C09025=1038.692,60.769,-88.501,169.467,39.132,157.356
C09026=1038.685,60.483,-88.481,169.465,39.132,157.356
C09027=1038.677,60.197,-88.461,169.463,39.132,157.356
C09028=1038.672,59.947,-88.444,169.461,39.131,157.356
C09029=1038.665,59.698,-88.426,169.459,39.131,157.356
C09030=1038.659,59.448,-88.409,169.457,39.131,157.356
C09031=1038.652,59.200,-88.392,169.454,39.130,157.356
C09032=1038.645,58.951,-88.373,169.452,39.130,157.356
C09033=1038.639,58.701,-88.356,169.450,39.130,157.355
C09034=1038.633,58.452,-88.339,169.448,39.129,157.355
C09035=1038.627,58.203,-88.321,169.446,39.130,157.355
C09036=1038.620,57.953,-88.303,169.444,39.129,157.355
C09037=1038.614,57.704,-88.286,169.442,39.129,157.355
C09038=1038.607,57.455,-88.268,169.440,39.128,157.355
C09039=1038.601,57.205,-88.251,169.438,39.128,157.355
C09040=1038.594,56.956,-88.234,169.436,39.128,157.355
C09041=1038.589,56.706,-88.217,169.433,39.127,157.354
C09042=1038.582,56.457,-88.200,169.432,39.127,157.354
C09043=1038.575,56.208,-88.183,169.430,39.127,157.354
C09044=1038.569,55.958,-88.165,169.428,39.126,157.354
C09045=1038.562,55.709,-88.147,169.426,39.126,157.354
C09046=1038.557,55.460,-88.130,169.424,39.126,157.354
C09047=1038.550,55.210,-88.112,169.422,39.125,157.354
C09048=1038.544,54.962,-88.095,169.420,39.125,157.354
C09049=1038.538,54.712,-88.077,169.418,39.125,157.354
C09050=1038.531,54.462,-88.060,169.416,39.125,157.353
C09051=1038.525,54.214,-88.043,169.413,39.124,157.353
C09052=1038.518,53.964,-88.025,169.411,39.124,157.353
C09053=1038.512,53.715,-88.008,169.409,39.124,157.353
C09054=1038.506,53.465,-87.992,169.407,39.123,157.353
C09055=1038.500,53.216,-87.974,169.405,39.123,157.353
C09056=1038.493,52.967,-87.957,169.404,39.123,157.353
C09057=1038.486,52.717,-87.939,169.402,39.122,157.353
C09058=1038.481,52.468,-87.922,169.400,39.122,157.352
C09059=1038.474,52.219,-87.905,169.398,39.121,157.352
C09060=1038.468,51.970,-87.888,169.395,39.121,157.352
C09061=1038.462,51.720,-87.870,169.393,39.121,157.352
C09062=1038.456,51.471,-87.853,169.391,39.120,157.352
C09063=1038.449,51.222,-87.836,169.389,39.120,157.352
C09064=1038.443,50.973,-87.818,169.387,39.120,157.352
C09065=1038.437,50.723,-87.801,169.385,39.119,157.352
C09066=1038.431,50.474,-87.785,169.383,39.119,157.351
C09067=1038.424,50.224,-87.767,169.381,39.119,157.351
C09068=1038.418,49.975,-87.750,169.379,39.119,157.351
C09069=1038.411,49.726,-87.733,169.378,39.118,157.351
C09070=1038.406,49.475,-87.715,169.375,39.118,157.351
C09071=1038.399,49.227,-87.698,169.373,39.118,157.351
C09072=1038.393,48.978,-87.681,169.371,39.117,157.351
C09073=1038.387,48.728,-87.664,169.369,39.117,157.351
C09074=1038.381,48.479,-87.647,169.367,39.116,157.350
C09075=1038.374,48.230,-87.630,169.365,39.116,157.350
C09076=1038.369,47.980,-87.612,169.363,39.116,157.350
C09077=1038.362,47.731,-87.595,169.361,39.115,157.350
C09078=1038.356,47.482,-87.579,169.359,39.115,157.350
C09079=1038.350,47.232,-87.561,169.356,39.114,157.350
C09080=1038.343,46.983,-87.544,169.354,39.114,157.350
C09081=1038.337,46.733,-87.527,169.352,39.114,157.350
C09082=1038.331,46.484,-87.510,169.351,39.113,157.349
C09083=1038.324,46.235,-87.492,169.349,39.113,157.349
C09084=1038.318,45.985,-87.476,169.347,39.112,157.349
C09085=1038.312,45.737,-87.459,169.345,39.112,157.349
C09086=1038.306,45.487,-87.441,169.343,39.112,157.349
C09087=1038.300,45.238,-87.425,169.341,39.111,157.349
C09088=1038.293,44.951,-87.405,169.338,39.111,157.349
C09089=1038.286,44.664,-87.385,169.336,39.110,157.348
C09090=1038.279,44.378,-87.366,169.333,39.110,157.348
C09091=1038.271,44.091,-87.346,169.331,39.109,157.348
C09092=1038.266,43.842,-87.330,169.329,39.110,157.348
C09093=1038.259,43.592,-87.312,169.327,39.109,157.348
C09094=1038.253,43.343,-87.296,169.325,39.109,157.348
C09095=1038.247,43.094,-87.278,169.323,39.108,157.348
C09096=1038.241,42.845,-87.261,169.321,39.108,157.348
C09097=1038.235,42.595,-87.245,169.319,39.108,157.347
C09098=1038.228,42.346,-87.227,169.317,39.107,157.347
C09099=1038.222,42.096,-87.211,169.315,39.107,157.347
C09100=1038.215,41.846,-87.195,169.313,39.107,157.347
C09101=1038.209,41.598,-87.178,169.311,39.106,157.347
C09102=1038.203,41.348,-87.161,169.309,39.106,157.347
C09103=1038.196,41.099,-87.144,169.307,39.106,157.347
C09104=1038.190,40.849,-87.128,169.305,39.105,157.347
C09105=1038.183,40.600,-87.110,169.303,39.105,157.347
C09106=1038.177,40.351,-87.094,169.301,39.105,157.346
C09107=1038.171,40.102,-87.077,169.298,39.104,157.346
C09108=1038.165,39.852,-87.061,169.296,39.105,157.346
C09109=1038.159,39.603,-87.044,169.294,39.104,157.346
C09110=1038.152,39.354,-87.027,169.292,39.104,157.346
C09111=1038.146,39.104,-87.011,169.290,39.104,157.346
C09112=1038.140,38.855,-86.994,169.288,39.103,157.346
C09113=1038.133,38.605,-86.977,169.286,39.103,157.346
C09114=1038.127,38.356,-86.961,169.284,39.103,157.346
C09115=1038.121,38.107,-86.944,169.282,39.102,157.345
C09116=1038.114,37.857,-86.927,169.279,39.102,157.345
C09117=1038.108,37.608,-86.911,169.277,39.102,157.345
C09118=1038.102,37.359,-86.894,169.275,39.101,157.345
C09119=1038.096,37.109,-86.877,169.273,39.101,157.345
C09120=1038.090,36.859,-86.861,169.271,39.101,157.345
C09121=1038.083,36.611,-86.844,169.269,39.101,157.345
C09122=1038.076,36.361,-86.828,169.267,39.101,157.345
C09123=1038.070,36.112,-86.812,169.265,39.100,157.344
C09124=1038.064,35.862,-86.796,169.263,39.100,157.344
C09125=1038.057,35.613,-86.778,169.261,39.100,157.344
C09126=1038.051,35.363,-86.762,169.259,39.099,157.344
C09127=1038.045,35.114,-86.746,169.257,39.099,157.344
C09128=1038.038,34.864,-86.730,169.255,39.099,157.344
C09129=1038.032,34.616,-86.713,169.253,39.099,157.344
C09130=1038.026,34.366,-86.697,169.251,39.099,157.344
C09131=1038.019,34.116,-86.680,169.249,39.098,157.344
C09132=1038.013,33.867,-86.664,169.247,39.098,157.344
C09133=1038.007,33.618,-86.648,169.245,39.098,157.343
C09134=1038.000,33.368,-86.631,169.243,39.098,157.343
C09135=1037.994,33.119,-86.614,169.241,39.097,157.343
C09136=1037.988,32.870,-86.598,169.239,39.097,157.343
C09137=1037.981,32.620,-86.582,169.237,39.097,157.343
C09138=1037.975,32.371,-86.566,169.235,39.096,157.343
C09139=1037.969,32.121,-86.550,169.233,39.097,157.343
C09140=1037.962,31.873,-86.533,169.230,39.096,157.343
C09141=1037.956,31.623,-86.516,169.228,39.095,157.343
C09142=1037.949,31.374,-86.500,169.226,39.096,157.342
C09143=1037.943,31.124,-86.484,169.224,39.095,157.342
C09144=1037.937,30.875,-86.468,169.222,39.095,157.342
C09145=1037.931,30.625,-86.451,169.220,39.095,157.342
C09146=1037.924,30.376,-86.436,169.218,39.094,157.342
C09147=1037.918,30.126,-86.419,169.216,39.094,157.342
C09148=1037.912,29.877,-86.403,169.214,39.094,157.342
C09149=1037.906,29.627,-86.386,169.212,39.094,157.342
C09150=1037.899,29.379,-86.370,169.210,39.093,157.342
C09151=1037.893,29.129,-86.354,169.207,39.093,157.341
C09152=1037.886,28.842,-86.336,169.204,39.093,157.341
C09153=1037.879,28.556,-86.317,169.202,39.093,157.341
C09154=1037.871,28.269,-86.298,169.200,39.092,157.341
C09155=1037.864,27.982,-86.280,169.197,39.092,157.341
C09156=1037.858,27.733,-86.263,169.195,39.092,157.341
C09157=1037.851,27.484,-86.248,169.193,39.092,157.341
C09158=1037.845,27.234,-86.231,169.191,39.091,157.341
C09159=1037.839,26.984,-86.215,169.189,39.091,157.341
C09160=1037.832,26.735,-86.199,169.187,39.091,157.340
C09161=1037.826,26.486,-86.183,169.184,39.091,157.340
C09162=1037.819,26.237,-86.167,169.182,39.091,157.340
C09163=1037.813,25.987,-86.151,169.180,39.090,157.340
C09164=1037.806,25.738,-86.135,169.178,39.090,157.340
C09165=1037.800,25.488,-86.119,169.176,39.090,157.340
C09166=1037.794,25.239,-86.102,169.174,39.090,157.340
C09167=1037.788,24.989,-86.088,169.172,39.089,157.340
C09168=1037.781,24.739,-86.071,169.170,39.090,157.340
C09169=1037.775,24.490,-86.055,169.168,39.089,157.340
C09170=1037.769,24.241,-86.039,169.166,39.089,157.340
C09171=1037.762,23.992,-86.023,169.164,39.089,157.339
C09172=1037.756,23.742,-86.007,169.162,39.089,157.339
C09173=1037.749,23.493,-85.991,169.160,39.088,157.339
C09174=1037.743,23.243,-85.976,169.158,39.088,157.339
C09175=1037.736,22.994,-85.960,169.155,39.088,157.339
C09176=1037.730,22.744,-85.944,169.153,39.088,157.339
C09177=1037.724,22.495,-85.928,169.151,39.088,157.339
C09178=1037.718,22.246,-85.912,169.149,39.088,157.339
C09179=1037.711,21.997,-85.896,169.147,39.087,157.339
C09180=1037.705,21.747,-85.880,169.145,39.087,157.338
C09181=1037.699,21.498,-85.865,169.143,39.087,157.338
C09182=1037.692,21.248,-85.848,169.141,39.086,157.338
C09183=1037.686,20.999,-85.833,169.139,39.086,157.338
C09184=1037.680,20.749,-85.817,169.137,39.086,157.338
C09185=1037.673,20.500,-85.801,169.135,39.086,157.338
C09186=1037.667,20.251,-85.785,169.133,39.086,157.338
C09187=1037.661,20.001,-85.769,169.129,39.086,157.338
C09188=1037.655,19.752,-85.754,169.127,39.085,157.338
C09189=1037.648,19.502,-85.738,169.125,39.085,157.338
C09190=1037.642,19.253,-85.722,169.123,39.085,157.338
C09191=1037.635,19.003,-85.707,169.121,39.085,157.337
C09192=1037.629,18.753,-85.690,169.119,39.084,157.337
C09193=1037.623,18.504,-85.675,169.117,39.085,157.337
C09194=1037.616,18.255,-85.660,169.115,39.084,157.337
C09195=1037.610,18.005,-85.644,169.113,39.084,157.337
C09196=1037.604,17.756,-85.628,169.111,39.084,157.337
C09197=1037.597,17.507,-85.613,169.109,39.084,157.337
C09198=1037.591,17.257,-85.597,169.107,39.083,157.337
C09199=1037.585,17.008,-85.581,169.105,39.083,157.337
C09200=1037.578,16.759,-85.566,169.102,39.083,157.337
C09201=1037.572,16.509,-85.550,169.100,39.083,157.337
C09202=1037.566,16.260,-85.535,169.098,39.083,157.336
C09203=1037.560,16.010,-85.519,169.096,39.083,157.336
C09204=1037.553,15.761,-85.503,169.093,39.082,157.336
C09205=1037.547,15.512,-85.488,169.091,39.082,157.336
C09206=1037.541,15.262,-85.472,169.089,39.082,157.336
C09207=1037.535,15.013,-85.457,169.087,39.082,157.336
C09208=1037.527,14.763,-85.441,169.085,39.082,157.336
C09209=1037.522,14.513,-85.425,169.083,39.082,157.336
C09210=1037.515,14.264,-85.410,169.081,39.082,157.336
C09211=1037.509,14.014,-85.395,169.079,39.081,157.336
C09212=1037.503,13.765,-85.378,169.077,39.081,157.336
C09213=1037.496,13.515,-85.363,169.074,39.081,157.335
C09214=1037.490,13.266,-85.348,169.072,39.081,157.335
C09215=1037.483,13.016,-85.333,169.070,39.081,157.335
C09216=1037.476,12.731,-85.315,169.067,39.081,157.335
C09217=1037.468,12.446,-85.297,169.065,39.081,157.335
C09218=1037.461,12.161,-85.280,169.062,39.080,157.335
C09219=1037.454,11.876,-85.263,169.060,39.081,157.335
C09220=1037.447,11.626,-85.247,169.058,39.081,157.335
C09221=1037.440,11.376,-85.232,169.056,39.080,157.335
C09222=1037.434,11.127,-85.217,169.054,39.080,157.335
C09223=1037.428,10.877,-85.201,169.051,39.081,157.335
C09224=1037.421,10.628,-85.186,169.049,39.080,157.334
C09225=1037.415,10.379,-85.171,169.047,39.080,157.334
C09226=1037.409,10.130,-85.156,169.045,39.080,157.334
C09227=1037.403,9.880,-85.141,169.043,39.080,157.334
C09228=1037.396,9.631,-85.125,169.041,39.080,157.334
C09229=1037.390,9.381,-85.110,169.038,39.079,157.334
C09230=1037.383,9.132,-85.095,169.036,39.080,157.334
C09231=1037.376,8.883,-85.080,169.033,39.080,157.334
C09232=1037.370,8.633,-85.065,169.031,39.079,157.334
C09233=1037.364,8.383,-85.050,169.029,39.079,157.334
C09234=1037.358,8.133,-85.034,169.027,39.079,157.334
C09235=1037.351,7.884,-85.019,169.025,39.079,157.334
C09236=1037.345,7.635,-85.004,169.023,39.079,157.334
C09237=1037.339,7.385,-84.989,169.021,39.079,157.333
C09238=1037.332,7.136,-84.973,169.019,39.079,157.333
C09239=1037.326,6.886,-84.958,169.017,39.079,157.333
C09240=1037.319,6.637,-84.943,169.014,39.078,157.333
C09241=1037.313,6.387,-84.928,169.012,39.079,157.333
C09242=1037.306,6.138,-84.912,169.010,39.079,157.333
C09243=1037.300,5.889,-84.898,169.008,39.078,157.333
C09244=1037.294,5.639,-84.883,169.006,39.078,157.333
C09245=1037.288,5.390,-84.868,169.003,39.078,157.333
C09246=1037.281,5.140,-84.853,169.001,39.078,157.333
C09247=1037.274,4.891,-84.837,168.999,39.078,157.333
C09248=1037.268,4.641,-84.822,168.996,39.078,157.332
C09249=1037.262,4.392,-84.808,168.994,39.078,157.332
C09250=1037.256,4.142,-84.792,168.992,39.077,157.332
C09251=1037.250,3.893,-84.777,168.990,39.077,157.332
C09252=1037.244,3.643,-84.762,168.988,39.077,157.332
C09253=1037.237,3.394,-84.747,168.986,39.077,157.332
C09254=1037.231,3.144,-84.732,168.984,39.077,157.332
C09255=1037.224,2.895,-84.717,168.981,39.077,157.332
C09256=1037.218,2.645,-84.702,168.979,39.077,157.332
C09257=1037.212,2.396,-84.687,168.977,39.077,157.332
C09258=1037.206,2.146,-84.672,168.975,39.076,157.332
C09259=1037.200,1.897,-84.657,168.973,39.077,157.332
C09260=1037.193,1.647,-84.643,168.970,39.076,157.331
C09261=1037.186,1.398,-84.627,168.968,39.076,157.331
C09262=1037.180,1.148,-84.612,168.966,39.076,157.331
C09263=1037.174,0.899,-84.597,168.963,39.076,157.331
C09264=1037.168,0.650,-84.582,168.961,39.076,157.331
C09265=1037.162,0.400,-84.567,168.959,39.075,157.331
C09266=1037.155,0.151,-84.552,168.957,39.076,157.331
C09267=1037.149,-0.098,-84.538,168.955,39.076,157.331
C09268=1037.143,-0.348,-84.523,168.953,39.075,157.331
C09269=1037.137,-0.598,-84.508,168.951,39.075,157.331
C09270=1037.130,-0.847,-84.493,168.948,39.075,157.331
C09271=1037.124,-1.097,-84.478,168.946,39.075,157.331
C09272=1037.118,-1.346,-84.464,168.944,39.075,157.331
C09273=1037.112,-1.596,-84.449,168.942,39.075,157.330
C09274=1037.105,-1.845,-84.434,168.940,39.075,157.330
C09275=1037.099,-2.094,-84.419,168.938,39.074,157.330
C09276=1037.093,-2.344,-84.404,168.935,39.074,157.330
C09277=1037.087,-2.594,-84.389,168.932,39.074,157.330
C09278=1037.080,-2.843,-84.374,168.930,39.074,157.330
C09279=1037.075,-3.092,-84.360,168.928,39.074,157.330
C09280=1037.068,-3.377,-84.342,168.926,39.074,157.330
C09281=1037.060,-3.660,-84.325,168.923,39.074,157.330
C09282=1037.053,-3.943,-84.309,168.921,39.073,157.330
C09283=1037.046,-4.227,-84.293,168.918,39.074,157.329
C09284=1037.040,-4.476,-84.278,168.916,39.074,157.329
C09285=1037.033,-4.726,-84.263,168.914,39.074,157.329
C09286=1037.027,-4.975,-84.249,168.912,39.073,157.329
C09287=1037.021,-5.225,-84.234,168.909,39.074,157.329
C09288=1037.014,-5.474,-84.220,168.907,39.074,157.329
C09289=1037.007,-5.724,-84.205,168.905,39.074,157.329
C09290=1037.001,-5.973,-84.191,168.903,39.074,157.329
C09291=1036.995,-6.223,-84.177,168.901,39.073,157.329
C09292=1036.988,-6.472,-84.162,168.898,39.074,157.329
C09293=1036.982,-6.721,-84.147,168.896,39.074,157.329
C09294=1036.975,-6.971,-84.133,168.894,39.074,157.329
C09295=1036.969,-7.220,-84.118,168.891,39.073,157.329
C09296=1036.963,-7.471,-84.104,168.888,39.074,157.329
C09297=1036.956,-7.719,-84.090,168.886,39.074,157.329
C09298=1036.950,-7.969,-84.075,168.884,39.074,157.329
C09299=1036.944,-8.219,-84.061,168.882,39.073,157.328
C09300=1036.937,-8.468,-84.047,168.880,39.073,157.328
C09301=1036.931,-8.717,-84.032,168.877,39.074,157.328
C09302=1036.925,-8.967,-84.017,168.875,39.074,157.328
C09303=1036.918,-9.216,-84.004,168.873,39.074,157.328
C09304=1036.912,-9.466,-83.989,168.871,39.073,157.328
C09305=1036.906,-9.716,-83.974,168.868,39.074,157.328
C09306=1036.899,-9.965,-83.960,168.866,39.074,157.328
C09307=1036.893,-10.215,-83.945,168.864,39.074,157.328
C09308=1036.887,-10.464,-83.931,168.862,39.073,157.328
C09309=1036.880,-10.714,-83.917,168.860,39.073,157.328
C09310=1036.874,-10.963,-83.902,168.857,39.074,157.328
C09311=1036.869,-11.213,-83.888,168.855,39.074,157.328
C09312=1036.861,-11.462,-83.874,168.853,39.073,157.328
C09313=1036.855,-11.712,-83.859,168.851,39.073,157.328
C09314=1036.850,-11.961,-83.845,168.848,39.074,157.327
C09315=1036.842,-12.211,-83.831,168.846,39.074,157.327
C09316=1036.837,-12.460,-83.816,168.843,39.073,157.327
C09317=1036.830,-12.710,-83.803,168.841,39.073,157.327
C09318=1036.823,-12.959,-83.788,168.839,39.074,157.327
C09319=1036.818,-13.209,-83.774,168.836,39.074,157.327
C09320=1036.811,-13.458,-83.760,168.834,39.073,157.327
C09321=1036.805,-13.708,-83.746,168.832,39.073,157.327
C09322=1036.799,-13.957,-83.731,168.830,39.073,157.327
C09323=1036.793,-14.207,-83.717,168.827,39.074,157.327
C09324=1036.786,-14.456,-83.703,168.825,39.073,157.327
C09325=1036.781,-14.706,-83.689,168.823,39.073,157.327
C09326=1036.774,-14.955,-83.674,168.821,39.073,157.327
C09327=1036.768,-15.206,-83.660,168.818,39.074,157.327
C09328=1036.761,-15.454,-83.646,168.816,39.073,157.326
C09329=1036.755,-15.704,-83.632,168.814,39.073,157.326
C09330=1036.749,-15.953,-83.618,168.812,39.073,157.326
C09331=1036.743,-16.203,-83.604,168.809,39.074,157.326
C09332=1036.736,-16.452,-83.590,168.807,39.074,157.326
C09333=1036.729,-16.702,-83.576,168.805,39.074,157.326
C09334=1036.723,-16.952,-83.562,168.802,39.074,157.326
C09335=1036.717,-17.201,-83.548,168.800,39.074,157.326
C09336=1036.710,-17.451,-83.534,168.798,39.074,157.326
C09337=1036.704,-17.700,-83.520,168.796,39.074,157.326
C09338=1036.697,-17.950,-83.506,168.793,39.074,157.326
C09339=1036.692,-18.199,-83.492,168.791,39.074,157.326
C09340=1036.685,-18.449,-83.478,168.788,39.074,157.326
C09341=1036.678,-18.698,-83.464,168.785,39.074,157.326
C09342=1036.672,-18.948,-83.450,168.783,39.075,157.326
C09343=1036.666,-19.197,-83.436,168.781,39.075,157.326
C09344=1036.659,-19.479,-83.421,168.778,39.075,157.326
C09345=1036.651,-19.761,-83.405,168.776,39.074,157.326
C09346=1036.644,-20.043,-83.390,168.773,39.075,157.325
C09347=1036.637,-20.325,-83.374,168.771,39.075,157.325
C09348=1036.631,-20.574,-83.360,168.768,39.075,157.325
C09349=1036.625,-20.824,-83.346,168.766,39.075,157.325
C09350=1036.618,-21.073,-83.332,168.764,39.075,157.325
C09351=1036.612,-21.323,-83.318,168.761,39.075,157.325
C09352=1036.606,-21.572,-83.305,168.759,39.076,157.325
C09353=1036.599,-21.822,-83.291,168.757,39.076,157.325
C09354=1036.593,-22.071,-83.276,168.754,39.075,157.325
C09355=1036.587,-22.321,-83.263,168.752,39.075,157.325
C09356=1036.580,-22.571,-83.250,168.750,39.075,157.325
C09357=1036.575,-22.820,-83.236,168.747,39.076,157.325
C09358=1036.568,-23.069,-83.221,168.745,39.076,157.325
C09359=1036.561,-23.319,-83.208,168.743,39.076,157.325
C09360=1036.555,-23.569,-83.194,168.741,39.076,157.325
C09361=1036.549,-23.818,-83.181,168.738,39.076,157.325
C09362=1036.543,-24.068,-83.167,168.736,39.076,157.325
C09363=1036.537,-24.318,-83.153,168.734,39.076,157.325
C09364=1036.530,-24.566,-83.139,168.731,39.076,157.325
C09365=1036.523,-24.816,-83.125,168.729,39.076,157.324
C09366=1036.518,-25.066,-83.112,168.727,39.076,157.324
C09367=1036.512,-25.315,-83.098,168.724,39.077,157.324
C09368=1036.505,-25.565,-83.085,168.722,39.077,157.324
C09369=1036.499,-25.815,-83.071,168.720,39.077,157.324
C09370=1036.493,-26.064,-83.058,168.717,39.077,157.324
C09371=1036.486,-26.314,-83.044,168.714,39.077,157.324
C09372=1036.481,-26.564,-83.030,168.712,39.077,157.324
C09373=1036.474,-26.812,-83.016,168.710,39.077,157.324
C09374=1036.468,-27.062,-83.002,168.707,39.077,157.324
C09375=1036.462,-27.312,-82.989,168.705,39.077,157.324
C09376=1036.455,-27.562,-82.975,168.702,39.077,157.324
C09377=1036.449,-27.811,-82.962,168.700,39.077,157.324
C09378=1036.443,-28.060,-82.948,168.698,39.078,157.324
C09379=1036.436,-28.310,-82.935,168.695,39.078,157.324
C09380=1036.430,-28.560,-82.921,168.693,39.078,157.324
C09381=1036.424,-28.809,-82.909,168.691,39.078,157.324
C09382=1036.417,-29.059,-82.895,168.688,39.078,157.324
C09383=1036.411,-29.309,-82.882,168.686,39.078,157.324
C09384=1036.405,-29.558,-82.869,168.684,39.079,157.324
C09385=1036.398,-29.808,-82.855,168.681,39.079,157.324
C09386=1036.392,-30.057,-82.842,168.679,39.079,157.324
C09387=1036.385,-30.306,-82.829,168.676,39.079,157.323
C09388=1036.379,-30.556,-82.815,168.674,39.079,157.323
C09389=1036.373,-30.806,-82.801,168.672,39.080,157.324
C09390=1036.367,-31.055,-82.788,168.669,39.080,157.323
C09391=1036.360,-31.305,-82.774,168.667,39.080,157.323
C09392=1036.354,-31.554,-82.761,168.665,39.080,157.323
C09393=1036.348,-31.804,-82.748,168.662,39.081,157.323
C09394=1036.341,-32.054,-82.735,168.660,39.081,157.323
C09395=1036.335,-32.304,-82.721,168.657,39.081,157.323
C09396=1036.329,-32.553,-82.708,168.655,39.081,157.323
C09397=1036.323,-32.802,-82.695,168.653,39.081,157.323
C09398=1036.316,-33.052,-82.681,168.650,39.081,157.323
C09399=1036.310,-33.302,-82.669,168.648,39.082,157.323
C09400=1036.304,-33.551,-82.655,168.645,39.082,157.323
C09401=1036.297,-33.800,-82.642,168.643,39.082,157.323
C09402=1036.291,-34.050,-82.629,168.641,39.082,157.323
C09403=1036.284,-34.300,-82.615,168.638,39.082,157.323
C09404=1036.278,-34.550,-82.603,168.636,39.082,157.323
C09405=1036.272,-34.799,-82.589,168.634,39.083,157.323
C09406=1036.265,-35.049,-82.576,168.631,39.083,157.323
C09407=1036.259,-35.298,-82.563,168.629,39.083,157.323
C09408=1036.251,-35.641,-82.544,168.625,39.083,157.323
C09409=1036.243,-35.985,-82.526,168.622,39.083,157.323
C09410=1036.234,-36.328,-82.508,168.619,39.084,157.323
C09411=1036.226,-36.672,-82.490,168.616,39.084,157.323
C09412=1036.220,-36.921,-82.477,168.613,39.084,157.323
C09413=1036.213,-37.171,-82.463,168.611,39.084,157.322
C09414=1036.207,-37.421,-82.451,168.608,39.084,157.322
C09415=1036.201,-37.670,-82.438,168.606,39.084,157.322
C09416=1036.195,-37.888,-82.426,168.604,39.085,157.322
C09417=1036.189,-38.107,-82.415,168.602,39.085,157.322
C09418=1036.184,-38.326,-82.404,168.600,39.085,157.322
C09419=1036.179,-38.544,-82.392,168.598,39.086,157.322
C09420=1036.174,-38.762,-82.380,168.596,39.086,157.322
C09421=1036.167,-38.981,-82.369,168.593,39.086,157.322
C09422=1036.162,-39.200,-82.358,168.591,39.086,157.322
C09423=1036.156,-39.418,-82.347,168.589,39.086,157.322
C09424=1036.150,-39.667,-82.334,168.587,39.086,157.322
C09425=1036.144,-39.917,-82.321,168.584,39.087,157.322
C09426=1036.138,-40.166,-82.308,168.582,39.087,157.322
C09427=1036.132,-40.416,-82.295,168.579,39.088,157.322
C09428=1036.125,-40.665,-82.282,168.577,39.088,157.322
C09429=1036.119,-40.915,-82.270,168.574,39.088,157.322
C09430=1036.112,-41.165,-82.256,168.572,39.088,157.322
C09431=1036.106,-41.415,-82.244,168.570,39.089,157.322
C09432=1036.100,-41.664,-82.231,168.567,39.089,157.322
C09433=1036.094,-41.914,-82.218,168.565,39.089,157.322
C09434=1036.087,-42.163,-82.205,168.562,39.089,157.322
C09435=1036.081,-42.413,-82.193,168.560,39.089,157.322
C09436=1036.075,-42.662,-82.180,168.557,39.090,157.322
C09437=1036.069,-42.912,-82.167,168.555,39.090,157.322
C09438=1036.062,-43.161,-82.154,168.552,39.091,157.322
C09439=1036.056,-43.411,-82.141,168.550,39.091,157.322
C09440=1036.049,-43.661,-82.129,168.547,39.091,157.322
C09441=1036.043,-43.910,-82.116,168.545,39.092,157.322
C09442=1036.037,-44.160,-82.103,168.542,39.092,157.322
C09443=1036.031,-44.409,-82.090,168.540,39.092,157.322
C09444=1036.024,-44.659,-82.078,168.538,39.092,157.322
C09445=1036.018,-44.909,-82.066,168.535,39.092,157.322
C09446=1036.012,-45.158,-82.052,168.533,39.093,157.322
C09447=1036.006,-45.408,-82.040,168.530,39.093,157.322
C09448=1035.999,-45.657,-82.027,168.528,39.094,157.322
C09449=1035.993,-45.907,-82.015,168.525,39.094,157.322
C09450=1035.987,-46.157,-82.002,168.523,39.094,157.322
C09451=1035.981,-46.406,-81.989,168.520,39.094,157.322
C09452=1035.975,-46.656,-81.977,168.518,39.095,157.322
C09453=1035.969,-46.905,-81.964,168.515,39.095,157.322
C09454=1035.962,-47.155,-81.951,168.513,39.095,157.322
C09455=1035.956,-47.404,-81.939,168.510,39.095,157.322
C09456=1035.950,-47.654,-81.926,168.508,39.096,157.322
C09457=1035.944,-47.904,-81.914,168.505,39.096,157.322
C09458=1035.938,-48.153,-81.901,168.503,39.097,157.322
C09459=1035.931,-48.403,-81.889,168.500,39.097,157.321
C09460=1035.925,-48.653,-81.876,168.498,39.097,157.321
C09461=1035.919,-48.902,-81.863,168.495,39.097,157.321
C09462=1035.912,-49.152,-81.851,168.493,39.098,157.321
C09463=1035.906,-49.401,-81.838,168.491,39.098,157.321
C09464=1035.901,-49.651,-81.826,168.488,39.098,157.321
C09465=1035.894,-49.901,-81.814,168.486,39.098,157.321
C09466=1035.888,-50.150,-81.801,168.483,39.099,157.321
C09467=1035.882,-50.400,-81.788,168.481,39.099,157.321
C09468=1035.875,-50.650,-81.776,168.478,39.100,157.321
C09469=1035.869,-50.900,-81.764,168.476,39.100,157.321
C09470=1035.863,-51.149,-81.752,168.473,39.101,157.321
C09471=1035.857,-51.399,-81.739,168.470,39.101,157.321
C09472=1035.849,-51.679,-81.726,168.468,39.102,157.321
C09473=1035.842,-51.961,-81.712,168.465,39.102,157.321
C09474=1035.835,-52.243,-81.697,168.462,39.103,157.321
C09475=1035.828,-52.524,-81.684,168.459,39.103,157.321
C09476=1035.822,-52.774,-81.672,168.456,39.104,157.321
C09477=1035.815,-53.023,-81.660,168.454,39.104,157.321
C09478=1035.809,-53.273,-81.648,168.451,39.105,157.321
C09479=1035.802,-53.523,-81.636,168.449,39.105,157.321
C09480=1035.796,-53.772,-81.624,168.446,39.106,157.322
C09481=1035.790,-54.022,-81.611,168.444,39.106,157.321
C09482=1035.783,-54.272,-81.599,168.441,39.106,157.321
C09483=1035.777,-54.521,-81.587,168.438,39.107,157.321
C09484=1035.771,-54.771,-81.575,168.436,39.107,157.321
C09485=1035.764,-55.021,-81.563,168.433,39.108,157.322
C09486=1035.757,-55.270,-81.551,168.431,39.108,157.321
C09487=1035.752,-55.520,-81.538,168.428,39.109,157.322
C09488=1035.745,-55.769,-81.527,168.426,39.109,157.322
C09489=1035.739,-56.019,-81.515,168.423,39.110,157.322
C09490=1035.733,-56.269,-81.502,168.420,39.110,157.322
C09491=1035.726,-56.518,-81.490,168.418,39.111,157.322
C09492=1035.720,-56.768,-81.478,168.415,39.111,157.322
C09493=1035.713,-57.017,-81.466,168.414,39.112,157.322
C09494=1035.707,-57.267,-81.454,168.410,39.112,157.322
C09495=1035.701,-57.517,-81.443,168.408,39.112,157.322
C09496=1035.695,-57.766,-81.431,168.406,39.113,157.322
C09497=1035.689,-58.016,-81.418,168.403,39.113,157.322
C09498=1035.682,-58.266,-81.406,168.401,39.114,157.322
C09499=1035.676,-58.515,-81.394,168.398,39.114,157.322
C09500=1035.670,-58.765,-81.382,168.396,39.115,157.322
C09501=1035.664,-59.014,-81.370,168.393,39.115,157.322
C09502=1035.657,-59.264,-81.359,168.391,39.116,157.322
C09503=1035.651,-59.514,-81.346,168.388,39.116,157.322
C09504=1035.645,-59.764,-81.334,168.385,39.117,157.322
C09505=1035.638,-60.013,-81.322,168.383,39.117,157.322
C09506=1035.632,-60.262,-81.311,168.380,39.118,157.322
C09507=1035.626,-60.513,-81.299,168.378,39.118,157.322
C09508=1035.620,-60.762,-81.287,168.375,39.119,157.322
C09509=1035.613,-61.012,-81.275,168.372,39.119,157.322
C09510=1035.608,-61.261,-81.263,168.370,39.119,157.322
C09511=1035.601,-61.511,-81.251,168.367,39.120,157.322
C09512=1035.595,-61.761,-81.240,168.365,39.120,157.322
C09513=1035.588,-62.010,-81.228,168.362,39.121,157.322
C09514=1035.583,-62.260,-81.216,168.360,39.121,157.322
C09515=1035.576,-62.510,-81.204,168.357,39.122,157.322
C09516=1035.570,-62.759,-81.192,168.354,39.123,157.322
C09517=1035.563,-63.009,-81.180,168.352,39.123,157.322
C09518=1035.558,-63.258,-81.168,168.349,39.124,157.322
C09519=1035.552,-63.508,-81.157,168.347,39.124,157.322
C09520=1035.545,-63.758,-81.145,168.344,39.125,157.322
C09521=1035.540,-64.007,-81.133,168.341,39.125,157.322
C09522=1035.533,-64.257,-81.122,168.339,39.126,157.322
C09523=1035.527,-64.507,-81.110,168.336,39.126,157.322
C09524=1035.520,-64.756,-81.098,168.334,39.127,157.322
C09525=1035.515,-65.006,-81.086,168.332,39.127,157.322
C09526=1035.508,-65.256,-81.074,168.329,39.128,157.322
C09527=1035.502,-65.506,-81.063,168.327,39.128,157.322
C09528=1035.496,-65.755,-81.051,168.324,39.129,157.322
C09529=1035.490,-66.005,-81.039,168.322,39.129,157.322
C09530=1035.484,-66.254,-81.028,168.319,39.130,157.322
C09531=1035.478,-66.504,-81.016,168.316,39.130,157.322
C09532=1035.471,-66.754,-81.005,168.314,39.131,157.322
C09533=1035.466,-67.003,-80.993,168.311,39.131,157.322
C09534=1035.459,-67.253,-80.981,168.309,39.132,157.322
C09535=1035.453,-67.503,-80.969,168.306,39.132,157.322
C09536=1035.446,-67.786,-80.956,168.303,39.133,157.322
C09537=1035.440,-68.068,-80.943,168.300,39.134,157.322
C09538=1035.433,-68.351,-80.930,168.297,39.134,157.322
C09539=1035.425,-68.634,-80.916,168.294,39.135,157.322
C09540=1035.419,-68.883,-80.905,168.292,39.135,157.322
C09541=1035.413,-69.133,-80.893,168.289,39.136,157.322
C09542=1035.408,-69.382,-80.882,168.286,39.136,157.322
C09543=1035.401,-69.632,-80.870,168.284,39.137,157.322
C09544=1035.395,-69.882,-80.859,168.281,39.137,157.322
C09545=1035.389,-70.131,-80.847,168.279,39.138,157.322
C09546=1035.384,-70.381,-80.836,168.276,39.138,157.322
C09547=1035.377,-70.631,-80.824,168.273,39.139,157.322
C09548=1035.371,-70.881,-80.813,168.271,39.139,157.322
C09549=1035.365,-71.130,-80.802,168.268,39.140,157.322
C09550=1035.358,-71.380,-80.790,168.265,39.140,157.322
C09551=1035.353,-71.630,-80.778,168.263,39.141,157.322
C09552=1035.347,-71.879,-80.766,168.260,39.141,157.322
C09553=1035.341,-72.129,-80.755,168.259,39.142,157.322
C09554=1035.335,-72.379,-80.744,168.256,39.143,157.322
C09555=1035.329,-72.628,-80.733,168.253,39.143,157.322
C09556=1035.323,-72.878,-80.721,168.251,39.144,157.322
C09557=1035.317,-73.128,-80.710,168.248,39.144,157.322
C09558=1035.311,-73.377,-80.698,168.245,39.145,157.322
C09559=1035.305,-73.627,-80.687,168.243,39.145,157.322
C09560=1035.298,-73.876,-80.675,168.240,39.146,157.322
C09561=1035.292,-74.126,-80.664,168.238,39.146,157.322
C09562=1035.286,-74.376,-80.653,168.235,39.147,157.322
C09563=1035.280,-74.625,-80.642,168.232,39.147,157.323
C09564=1035.274,-74.875,-80.630,168.230,39.148,157.322
C09565=1035.268,-75.125,-80.619,168.227,39.148,157.323
C09566=1035.262,-75.375,-80.608,168.224,39.149,157.323
C09567=1035.256,-75.624,-80.597,168.222,39.149,157.323
C09568=1035.250,-75.874,-80.586,168.219,39.150,157.323
C09569=1035.244,-76.123,-80.574,168.216,39.151,157.323
C09570=1035.237,-76.373,-80.563,168.213,39.152,157.323
C09571=1035.231,-76.623,-80.552,168.211,39.152,157.323
C09572=1035.226,-76.872,-80.541,168.209,39.153,157.323
C09573=1035.219,-77.122,-80.531,168.206,39.154,157.323
C09574=1035.213,-77.371,-80.519,168.204,39.155,157.323
C09575=1035.206,-77.621,-80.508,168.201,39.155,157.323
C09576=1035.200,-77.871,-80.497,168.198,39.156,157.323
C09577=1035.194,-78.121,-80.486,168.196,39.157,157.323
C09578=1035.188,-78.371,-80.475,168.193,39.157,157.323
C09579=1035.183,-78.620,-80.464,168.190,39.158,157.323
C09580=1035.176,-78.870,-80.453,168.188,39.159,157.323
C09581=1035.171,-79.120,-80.442,168.185,39.159,157.323
C09582=1035.164,-79.369,-80.430,168.182,39.160,157.323
C09583=1035.158,-79.619,-80.419,168.180,39.160,157.323
C09584=1035.151,-79.869,-80.408,168.177,39.161,157.323
C09585=1035.145,-80.118,-80.397,168.174,39.162,157.323
C09586=1035.140,-80.368,-80.387,168.171,39.163,157.323
C09587=1035.133,-80.618,-80.376,168.170,39.164,157.323
C09588=1035.127,-80.867,-80.365,168.167,39.164,157.323
C09589=1035.120,-81.117,-80.354,168.164,39.165,157.323
C09590=1035.114,-81.366,-80.343,168.161,39.166,157.324
C09591=1035.108,-81.616,-80.333,168.159,39.167,157.324
C09592=1035.102,-81.866,-80.321,168.156,39.167,157.324
C09593=1035.095,-82.115,-80.311,168.153,39.168,157.324
C09594=1035.089,-82.366,-80.301,168.150,39.169,157.324
C09595=1035.084,-82.616,-80.290,168.148,39.170,157.324
C09596=1035.077,-82.865,-80.279,168.145,39.171,157.324
C09597=1035.071,-83.115,-80.268,168.142,39.172,157.324
C09598=1035.065,-83.364,-80.257,168.140,39.172,157.324
C09599=1035.059,-83.614,-80.247,168.138,39.173,157.324
C09600=1035.051,-83.899,-80.235,168.135,39.174,157.324
C09601=1035.045,-84.184,-80.223,168.132,39.175,157.324
C09602=1035.037,-84.469,-80.210,168.128,39.176,157.324
C09603=1035.030,-84.753,-80.198,168.125,39.177,157.324
C09604=1035.024,-85.004,-80.187,168.122,39.178,157.324
///RCONF 1,0,0,0,1,0,0,0,0,0,0,0,0,0,0,0,0,0,0,0,0,0,0,0
C09605=1035.018,-85.253,-80.177,168.120,39.179,157.325
C09606=1035.012,-85.502,-80.166,168.117,39.179,157.325
C09607=1035.006,-85.753,-80.155,168.114,39.180,157.325
C09608=1034.999,-86.002,-80.145,168.111,39.181,157.325
C09609=1034.993,-86.251,-80.134,168.109,39.181,157.325
C09610=1034.988,-86.501,-80.124,168.106,39.182,157.325
C09611=1034.981,-86.751,-80.113,168.104,39.183,157.325
C09612=1034.975,-87.001,-80.102,168.101,39.184,157.325
C09613=1034.969,-87.250,-80.092,168.099,39.185,157.325
C09614=1034.963,-87.501,-80.081,168.096,39.186,157.325
C09615=1034.957,-87.750,-80.070,168.093,39.187,157.325
C09616=1034.950,-87.999,-80.060,168.090,39.187,157.325
C09617=1034.945,-88.249,-80.049,168.088,39.188,157.325
C09618=1034.939,-88.499,-80.040,168.085,39.189,157.325
C09619=1034.932,-88.749,-80.028,168.082,39.190,157.325
C09620=1034.926,-88.998,-80.017,168.079,39.191,157.325
C09621=1034.920,-89.248,-80.007,168.078,39.192,157.326
C09622=1034.915,-89.498,-79.997,168.075,39.192,157.326
C09623=1034.907,-89.748,-79.986,168.072,39.193,157.326
C09624=1034.902,-89.997,-79.976,168.069,39.194,157.326
C09625=1034.896,-90.247,-79.965,168.067,39.195,157.326
C09626=1034.890,-90.496,-79.955,168.064,39.196,157.326
C09627=1034.884,-90.746,-79.944,168.061,39.197,157.326
C09628=1034.877,-90.996,-79.934,168.058,39.198,157.326
C09629=1034.872,-91.246,-79.923,168.056,39.198,157.326
C09630=1034.865,-91.495,-79.913,168.053,39.199,157.326
C09631=1034.860,-91.745,-79.903,168.050,39.200,157.326
C09632=1034.854,-91.995,-79.892,168.048,39.201,157.326
C09633=1034.848,-92.244,-79.882,168.046,39.202,157.326
C09634=1034.842,-92.494,-79.872,168.043,39.203,157.326
C09635=1034.835,-92.744,-79.861,168.040,39.204,157.326
C09636=1034.829,-92.994,-79.851,168.037,39.204,157.327
C09637=1034.823,-93.243,-79.841,168.034,39.205,157.327
C09638=1034.818,-93.493,-79.830,168.032,39.206,157.327
C09639=1034.812,-93.743,-79.819,168.029,39.206,157.327
C09640=1034.806,-93.992,-79.810,168.026,39.207,157.327
C09641=1034.800,-94.242,-79.799,168.023,39.208,157.327
C09642=1034.794,-94.492,-79.789,168.021,39.209,157.327
C09643=1034.787,-94.742,-79.778,168.018,39.210,157.327
C09644=1034.781,-94.992,-79.769,168.016,39.211,157.327
C09645=1034.775,-95.241,-79.758,168.013,39.212,157.327
C09646=1034.769,-95.491,-79.748,168.010,39.212,157.327
C09647=1034.764,-95.741,-79.737,168.008,39.213,157.327
C09648=1034.757,-95.990,-79.728,168.005,39.215,157.327
C09649=1034.752,-96.240,-79.717,168.002,39.216,157.327
C09650=1034.745,-96.490,-79.707,167.999,39.217,157.327
C09651=1034.740,-96.739,-79.696,167.997,39.217,157.327
C09652=1034.734,-96.989,-79.686,167.994,39.218,157.328
C09653=1034.728,-97.238,-79.676,167.992,39.219,157.328
C09654=1034.722,-97.488,-79.666,167.989,39.220,157.328
C09655=1034.716,-97.738,-79.656,167.986,39.221,157.328
C09656=1034.710,-97.987,-79.646,167.984,39.222,157.328
C09657=1034.704,-98.238,-79.636,167.981,39.223,157.328
C09658=1034.698,-98.487,-79.626,167.978,39.223,157.328
C09659=1034.691,-98.737,-79.616,167.975,39.225,157.328
C09660=1034.685,-98.987,-79.606,167.972,39.226,157.328
C09661=1034.679,-99.237,-79.596,167.970,39.227,157.328
C09662=1034.673,-99.486,-79.586,167.967,39.228,157.328
C09663=1034.667,-99.736,-79.576,167.965,39.228,157.328
C09664=1034.661,-100.023,-79.565,167.962,39.230,157.329
C09665=1034.654,-100.310,-79.553,167.958,39.231,157.329
C09666=1034.646,-100.598,-79.542,167.955,39.232,157.329
C09667=1034.640,-100.885,-79.530,167.952,39.233,157.329
C09668=1034.633,-101.134,-79.520,167.949,39.234,157.329
C09669=1034.627,-101.384,-79.510,167.946,39.235,157.329
C09670=1034.621,-101.634,-79.501,167.944,39.237,157.329
C09671=1034.615,-101.884,-79.491,167.942,39.237,157.329
C09672=1034.609,-102.133,-79.480,167.939,39.238,157.329
C09673=1034.603,-102.382,-79.471,167.936,39.239,157.329
C09674=1034.597,-102.632,-79.462,167.933,39.241,157.330
C09675=1034.592,-102.882,-79.451,167.930,39.242,157.330
C09676=1034.586,-103.132,-79.442,167.927,39.242,157.330
C09677=1034.579,-103.381,-79.432,167.925,39.243,157.330
C09678=1034.573,-103.631,-79.422,167.922,39.244,157.330
C09679=1034.568,-103.881,-79.412,167.920,39.246,157.330
C09680=1034.561,-104.131,-79.402,167.917,39.247,157.330
C09681=1034.555,-104.381,-79.393,167.914,39.247,157.330
C09682=1034.549,-104.631,-79.383,167.911,39.249,157.330
C09683=1034.543,-104.880,-79.374,167.909,39.250,157.330
C09684=1034.537,-105.131,-79.363,167.906,39.251,157.330
C09685=1034.531,-105.380,-79.353,167.903,39.252,157.330
C09686=1034.525,-105.630,-79.344,167.901,39.253,157.331
C09687=1034.519,-105.879,-79.334,167.898,39.254,157.331
C09688=1034.513,-106.128,-79.325,167.895,39.255,157.331
C09689=1034.508,-106.379,-79.315,167.892,39.256,157.331
C09690=1034.501,-106.628,-79.305,167.890,39.257,157.331
C09691=1034.495,-106.878,-79.296,167.887,39.258,157.331
C09692=1034.489,-107.128,-79.286,167.884,39.259,157.331
C09693=1034.483,-107.378,-79.276,167.881,39.261,157.331
C09694=1034.477,-107.628,-79.267,167.878,39.261,157.331
C09695=1034.472,-107.877,-79.257,167.876,39.262,157.331
C09696=1034.466,-108.127,-79.247,167.873,39.264,157.332
C09697=1034.460,-108.377,-79.238,167.871,39.265,157.332
C09698=1034.453,-108.626,-79.228,167.868,39.266,157.332
C09699=1034.447,-108.876,-79.219,167.865,39.267,157.332
C09700=1034.441,-109.126,-79.209,167.862,39.268,157.332
C09701=1034.435,-109.376,-79.200,167.859,39.270,157.332
C09702=1034.430,-109.625,-79.191,167.857,39.270,157.332
C09703=1034.423,-109.875,-79.182,167.854,39.272,157.332
C09704=1034.417,-110.125,-79.172,167.851,39.273,157.332
C09705=1034.411,-110.375,-79.162,167.849,39.274,157.333
C09706=1034.405,-110.625,-79.153,167.846,39.275,157.333
C09707=1034.399,-110.874,-79.144,167.843,39.276,157.333
C09708=1034.393,-111.124,-79.134,167.841,39.278,157.333
C09709=1034.387,-111.373,-79.125,167.838,39.279,157.333
C09710=1034.381,-111.624,-79.116,167.835,39.280,157.333
C09711=1034.375,-111.874,-79.106,167.832,39.281,157.333
C09712=1034.369,-112.123,-79.097,167.829,39.282,157.333
C09713=1034.363,-112.372,-79.087,167.827,39.283,157.333
C09714=1034.357,-112.622,-79.078,167.824,39.284,157.334
C09715=1034.351,-112.872,-79.068,167.822,39.286,157.334
C09716=1034.346,-113.122,-79.060,167.819,39.287,157.334
C09717=1034.339,-113.372,-79.050,167.816,39.288,157.334
C09718=1034.333,-113.621,-79.041,167.813,39.289,157.334
C09719=1034.327,-113.871,-79.031,167.810,39.291,157.334
C09720=1034.322,-114.121,-79.023,167.807,39.292,157.334
C09721=1034.316,-114.371,-79.013,167.804,39.292,157.334
C09722=1034.309,-114.620,-79.003,167.803,39.294,157.335
C09723=1034.303,-114.870,-78.994,167.800,39.295,157.335
C09724=1034.298,-115.120,-78.985,167.797,39.296,157.335
C09725=1034.292,-115.370,-78.976,167.794,39.298,157.335
C09726=1034.286,-115.620,-78.966,167.791,39.299,157.335
C09727=1034.280,-115.869,-78.958,167.788,39.300,157.335
C09728=1034.273,-116.156,-78.947,167.785,39.301,157.335
C09729=1034.266,-116.442,-78.937,167.782,39.303,157.335
C09730=1034.259,-116.728,-78.926,167.779,39.304,157.336
C09731=1034.252,-117.015,-78.915,167.776,39.306,157.336
C09732=1034.246,-117.266,-78.907,167.773,39.307,157.336
C09733=1034.241,-117.515,-78.897,167.770,39.308,157.336
C09734=1034.234,-117.764,-78.888,167.767,39.309,157.336
C09735=1034.229,-118.015,-78.879,167.765,39.311,157.336
C09736=1034.222,-118.264,-78.870,167.762,39.312,157.336
C09737=1034.216,-118.514,-78.862,167.759,39.313,157.336
C09738=1034.210,-118.764,-78.852,167.756,39.315,157.337
C09739=1034.205,-119.014,-78.843,167.753,39.316,157.337
C09740=1034.199,-119.263,-78.834,167.751,39.317,157.337
C09741=1034.193,-119.512,-78.825,167.749,39.319,157.337
C09742=1034.187,-119.763,-78.816,167.746,39.320,157.337
C09743=1034.181,-120.012,-78.807,167.743,39.321,157.337
C09744=1034.175,-120.262,-78.798,167.740,39.322,157.337
C09745=1034.169,-120.512,-78.789,167.737,39.324,157.337
C09746=1034.164,-120.762,-78.780,167.735,39.325,157.338
C09747=1034.157,-121.011,-78.771,167.732,39.326,157.338
C09748=1034.151,-121.261,-78.763,167.729,39.328,157.338
C09749=1034.145,-121.511,-78.753,167.726,39.329,157.338
C09750=1034.140,-121.761,-78.744,167.723,39.330,157.338
C09751=1034.133,-122.010,-78.736,167.720,39.332,157.338
C09752=1034.127,-122.260,-78.727,167.718,39.333,157.338
C09753=1034.122,-122.511,-78.718,167.716,39.334,157.339
C09754=1034.116,-122.760,-78.709,167.713,39.336,157.339
C09755=1034.110,-123.010,-78.700,167.710,39.337,157.339
C09756=1034.104,-123.259,-78.692,167.707,39.338,157.339
C09757=1034.098,-123.509,-78.683,167.704,39.340,157.339
C09758=1034.093,-123.759,-78.674,167.701,39.341,157.339
C09759=1034.087,-124.009,-78.665,167.699,39.342,157.339
C09760=1034.081,-124.258,-78.657,167.696,39.344,157.340
C09761=1034.074,-124.508,-78.647,167.693,39.345,157.340
C09762=1034.069,-124.758,-78.639,167.690,39.346,157.340
C09763=1034.062,-125.008,-78.630,167.687,39.348,157.340
C09764=1034.056,-125.258,-78.621,167.685,39.349,157.340
C09765=1034.051,-125.507,-78.612,167.682,39.350,157.340
C09766=1034.044,-125.757,-78.604,167.679,39.352,157.340
C09767=1034.039,-126.007,-78.596,167.676,39.353,157.341
C09768=1034.032,-126.257,-78.587,167.674,39.355,157.341
C09769=1034.027,-126.506,-78.578,167.672,39.356,157.341
C09770=1034.021,-126.757,-78.569,167.669,39.357,157.341
C09771=1034.015,-127.006,-78.561,167.666,39.359,157.341
C09772=1034.010,-127.255,-78.552,167.663,39.360,157.341
C09773=1034.003,-127.505,-78.544,167.660,39.362,157.341
C09774=1033.997,-127.754,-78.535,167.657,39.363,157.342
C09775=1033.992,-128.004,-78.526,167.655,39.364,157.342
C09776=1033.987,-128.254,-78.516,167.652,39.365,157.342
C09777=1033.983,-128.504,-78.507,167.650,39.365,157.342
C09778=1033.979,-128.754,-78.496,167.647,39.365,157.342
C09779=1033.977,-129.004,-78.485,167.644,39.364,157.341
C09780=1033.974,-129.253,-78.473,167.642,39.363,157.341
C09781=1033.973,-129.503,-78.461,167.641,39.362,157.341
C09782=1033.972,-129.753,-78.448,167.638,39.360,157.340
C09783=1033.972,-130.003,-78.434,167.637,39.357,157.340
C09784=1033.973,-130.253,-78.420,167.634,39.354,157.339
C09785=1033.974,-130.503,-78.405,167.633,39.351,157.339
C09786=1033.976,-130.753,-78.390,167.631,39.347,157.338
C09787=1033.978,-131.002,-78.374,167.630,39.343,157.337
C09788=1033.982,-131.253,-78.358,167.628,39.338,157.336
C09789=1033.986,-131.503,-78.341,167.627,39.333,157.336
C09790=1033.992,-131.753,-78.323,167.626,39.327,157.334
C09791=1033.997,-132.003,-78.305,167.625,39.321,157.333
C09792=1033.666,-132.027,-78.591,167.576,39.544,157.369
C09793=1033.661,-131.778,-78.609,167.577,39.550,157.370
C09794=1033.656,-131.528,-78.626,167.579,39.555,157.371
C09795=1033.652,-131.278,-78.643,167.580,39.561,157.372
C09796=1033.648,-131.028,-78.660,167.581,39.565,157.373
C09797=1033.646,-130.778,-78.676,167.583,39.570,157.374
C09798=1033.644,-130.527,-78.691,167.584,39.574,157.375
C09799=1033.643,-130.278,-78.706,167.586,39.577,157.375
C09800=1033.642,-130.027,-78.720,167.588,39.580,157.376
C09801=1033.642,-129.777,-78.733,167.590,39.583,157.376
C09802=1033.643,-129.528,-78.746,167.591,39.585,157.376
C09803=1033.644,-129.278,-78.759,167.594,39.586,157.377
C09804=1033.646,-129.028,-78.771,167.596,39.588,157.377
C09805=1033.648,-128.778,-78.782,167.598,39.588,157.377
C09806=1033.652,-128.528,-78.793,167.600,39.589,157.377
C09807=1033.657,-128.279,-78.803,167.603,39.588,157.377
C09808=1033.661,-128.029,-78.813,167.606,39.587,157.378
C09809=1033.667,-127.780,-78.821,167.609,39.586,157.377
C09810=1033.673,-127.530,-78.829,167.611,39.584,157.377
C09811=1033.679,-127.280,-78.839,167.614,39.583,157.377
C09812=1033.684,-127.031,-78.847,167.617,39.582,157.377
C09813=1033.690,-126.781,-78.855,167.619,39.580,157.377
C09814=1033.696,-126.531,-78.864,167.622,39.579,157.377
C09815=1033.702,-126.282,-78.873,167.625,39.577,157.376
C09816=1033.708,-126.032,-78.881,167.628,39.576,157.376
C09817=1033.713,-125.782,-78.890,167.631,39.575,157.376
C09818=1033.720,-125.533,-78.899,167.633,39.573,157.376
C09819=1033.726,-125.283,-78.907,167.636,39.572,157.376
C09820=1033.731,-125.032,-78.916,167.639,39.570,157.376
C09821=1033.737,-124.783,-78.924,167.642,39.568,157.376
C09822=1033.744,-124.533,-78.934,167.645,39.567,157.375
C09823=1033.749,-124.283,-78.943,167.647,39.566,157.375
C09824=1033.755,-124.033,-78.950,167.650,39.564,157.375
C09825=1033.762,-123.784,-78.960,167.653,39.563,157.375
C09826=1033.767,-123.534,-78.968,167.656,39.562,157.375
C09827=1033.773,-123.284,-78.978,167.659,39.560,157.375
C09828=1033.779,-123.035,-78.986,167.662,39.559,157.375
C09829=1033.785,-122.784,-78.995,167.664,39.558,157.375
C09830=1033.790,-122.535,-79.004,167.667,39.556,157.374
C09831=1033.796,-122.285,-79.013,167.670,39.555,157.374
C09832=1033.803,-122.036,-79.021,167.673,39.553,157.374
C09833=1033.809,-121.786,-79.030,167.676,39.552,157.374
C09834=1033.815,-121.536,-79.040,167.678,39.551,157.374
C09835=1033.820,-121.286,-79.048,167.680,39.549,157.374
C09836=1033.827,-121.037,-79.057,167.683,39.548,157.374
C09837=1033.832,-120.787,-79.066,167.686,39.547,157.373
C09838=1033.838,-120.536,-79.075,167.689,39.545,157.373
C09839=1033.844,-120.287,-79.084,167.692,39.544,157.373
C09840=1033.849,-120.037,-79.093,167.694,39.542,157.373
C09841=1033.856,-119.787,-79.102,167.697,39.541,157.373
C09842=1033.862,-119.538,-79.111,167.700,39.540,157.373
C09843=1033.868,-119.288,-79.120,167.703,39.538,157.373
C09844=1033.874,-119.038,-79.129,167.706,39.538,157.373
C09845=1033.879,-118.788,-79.138,167.709,39.536,157.372
C09846=1033.885,-118.539,-79.147,167.711,39.534,157.372
C09847=1033.891,-118.289,-79.155,167.714,39.533,157.372
C09848=1033.898,-118.039,-79.165,167.717,39.532,157.372
C09849=1033.903,-117.789,-79.174,167.720,39.530,157.372
C09850=1033.909,-117.540,-79.183,167.723,39.529,157.372
C09851=1033.915,-117.290,-79.192,167.724,39.528,157.372
C09852=1033.921,-117.040,-79.201,167.727,39.526,157.371
C09853=1033.929,-116.753,-79.212,167.731,39.525,157.371
C09854=1033.935,-116.467,-79.222,167.734,39.524,157.371
C09855=1033.941,-116.181,-79.233,167.737,39.522,157.371
C09856=1033.948,-115.894,-79.243,167.741,39.521,157.371
C09857=1033.955,-115.644,-79.252,167.743,39.520,157.371
C09858=1033.961,-115.394,-79.262,167.746,39.518,157.371
C09859=1033.966,-115.145,-79.271,167.749,39.516,157.370
C09860=1033.972,-114.895,-79.280,167.751,39.516,157.370
C09861=1033.978,-114.645,-79.289,167.754,39.514,157.370
C09862=1033.984,-114.396,-79.298,167.757,39.513,157.370
C09863=1033.990,-114.145,-79.307,167.759,39.512,157.370
C09864=1033.996,-113.896,-79.317,167.762,39.511,157.370
C09865=1034.002,-113.646,-79.326,167.765,39.509,157.370
C09866=1034.008,-113.397,-79.336,167.768,39.508,157.370
C09867=1034.014,-113.146,-79.344,167.771,39.507,157.370
C09868=1034.020,-112.897,-79.354,167.774,39.506,157.369
C09869=1034.026,-112.647,-79.364,167.776,39.504,157.369
C09870=1034.032,-112.398,-79.373,167.779,39.503,157.369
C09871=1034.038,-112.148,-79.382,167.781,39.502,157.369
C09872=1034.044,-111.897,-79.391,167.784,39.501,157.369
C09873=1034.050,-111.648,-79.401,167.787,39.499,157.369
C09874=1034.055,-111.399,-79.410,167.790,39.498,157.369
C09875=1034.061,-111.149,-79.420,167.792,39.497,157.369
C09876=1034.068,-110.899,-79.429,167.795,39.496,157.369
C09877=1034.074,-110.649,-79.439,167.798,39.494,157.368
C09878=1034.080,-110.399,-79.448,167.801,39.493,157.368
C09879=1034.085,-110.150,-79.457,167.804,39.493,157.368
C09880=1034.091,-109.900,-79.466,167.807,39.491,157.368
C09881=1034.098,-109.650,-79.476,167.809,39.490,157.368
C09882=1034.104,-109.400,-79.485,167.811,39.489,157.368
C09883=1034.110,-109.150,-79.495,167.814,39.488,157.368
C09884=1034.116,-108.901,-79.504,167.817,39.486,157.368
C09885=1034.122,-108.652,-79.514,167.820,39.485,157.368
C09886=1034.128,-108.402,-79.523,167.823,39.484,157.367
C09887=1034.134,-108.152,-79.533,167.826,39.483,157.367
C09888=1034.140,-107.902,-79.543,167.829,39.481,157.367
C09889=1034.146,-107.652,-79.552,167.831,39.480,157.367
C09890=1034.153,-107.403,-79.562,167.834,39.479,157.367
C09891=1034.157,-107.153,-79.571,167.836,39.478,157.367
C09892=1034.164,-106.903,-79.581,167.839,39.477,157.367
C09893=1034.170,-106.654,-79.591,167.842,39.476,157.367
C09894=1034.176,-106.404,-79.600,167.845,39.475,157.367
C09895=1034.182,-106.154,-79.610,167.848,39.474,157.366
C09896=1034.188,-105.904,-79.619,167.850,39.472,157.366
C09897=1034.194,-105.654,-79.629,167.853,39.471,157.366
C09898=1034.200,-105.404,-79.639,167.856,39.470,157.366
C09899=1034.205,-105.155,-79.648,167.858,39.469,157.366
C09900=1034.212,-104.905,-79.658,167.861,39.468,157.366
C09901=1034.218,-104.656,-79.667,167.864,39.467,157.366
C09902=1034.223,-104.405,-79.677,167.867,39.466,157.366
C09903=1034.229,-104.156,-79.687,167.869,39.465,157.366
C09904=1034.236,-103.906,-79.697,167.872,39.464,157.366
C09905=1034.242,-103.657,-79.707,167.875,39.463,157.366
C09906=1034.247,-103.407,-79.717,167.877,39.461,157.365
C09907=1034.254,-103.157,-79.727,167.880,39.460,157.365
C09908=1034.260,-102.907,-79.736,167.883,39.459,157.365
C09909=1034.266,-102.657,-79.746,167.886,39.458,157.365
C09910=1034.271,-102.407,-79.756,167.889,39.457,157.365
C09911=1034.278,-102.158,-79.766,167.891,39.456,157.365
C09912=1034.284,-101.908,-79.776,167.894,39.455,157.365
C09913=1034.290,-101.658,-79.785,167.896,39.454,157.365
C09914=1034.296,-101.408,-79.796,167.899,39.453,157.365
C09915=1034.301,-101.159,-79.805,167.902,39.452,157.365
C09916=1034.308,-100.910,-79.815,167.905,39.451,157.365
C09917=1034.315,-100.623,-79.826,167.908,39.449,157.364
C09918=1034.322,-100.335,-79.838,167.911,39.449,157.364
C09919=1034.329,-100.048,-79.849,167.914,39.447,157.364
C09920=1034.336,-99.761,-79.860,167.917,39.446,157.364
C09921=1034.341,-99.511,-79.870,167.920,39.445,157.364
C09922=1034.348,-99.262,-79.881,167.923,39.444,157.364
C09923=1034.354,-99.012,-79.890,167.926,39.443,157.364
C09924=1034.360,-98.762,-79.900,167.928,39.442,157.364
C09925=1034.366,-98.513,-79.911,167.931,39.440,157.364
C09926=1034.372,-98.262,-79.921,167.933,39.439,157.364
C09927=1034.379,-98.012,-79.930,167.936,39.439,157.363
C09928=1034.384,-97.763,-79.941,167.939,39.438,157.363
C09929=1034.390,-97.513,-79.951,167.942,39.436,157.363
C09930=1034.397,-97.263,-79.960,167.944,39.435,157.363
C09931=1034.402,-97.014,-79.971,167.947,39.434,157.363
C09932=1034.408,-96.764,-79.981,167.950,39.433,157.363
C09933=1034.414,-96.515,-79.991,167.953,39.433,157.363
C09934=1034.420,-96.264,-80.002,167.956,39.432,157.363
C09935=1034.426,-96.015,-80.012,167.957,39.431,157.363
C09936=1034.432,-95.765,-80.022,167.960,39.430,157.363
C09937=1034.438,-95.515,-80.032,167.963,39.429,157.363
C09938=1034.444,-95.266,-80.043,167.966,39.428,157.363
C09939=1034.450,-95.016,-80.052,167.969,39.427,157.363
C09940=1034.455,-94.767,-80.063,167.971,39.426,157.363
C09941=1034.462,-94.517,-80.073,167.974,39.426,157.362
C09942=1034.467,-94.267,-80.083,167.977,39.425,157.362
C09943=1034.474,-94.017,-80.094,167.980,39.424,157.362
C09944=1034.480,-93.767,-80.104,167.983,39.423,157.362
C09945=1034.486,-93.518,-80.115,167.984,39.421,157.362
C09946=1034.492,-93.268,-80.125,167.987,39.421,157.362
C09947=1034.498,-93.018,-80.136,167.990,39.420,157.362
C09948=1034.504,-92.769,-80.145,167.993,39.419,157.362
C09949=1034.509,-92.519,-80.156,167.996,39.418,157.362
C09950=1034.516,-92.269,-80.166,167.998,39.417,157.362
C09951=1034.522,-92.019,-80.177,168.001,39.416,157.362
C09952=1034.528,-91.770,-80.187,168.004,39.415,157.362
C09953=1034.534,-91.520,-80.197,168.007,39.414,157.362
C09954=1034.540,-91.270,-80.208,168.009,39.414,157.362
C09955=1034.546,-91.021,-80.218,168.011,39.413,157.361
C09956=1034.552,-90.771,-80.229,168.014,39.412,157.361
C09957=1034.559,-90.521,-80.239,168.017,39.411,157.361
C09958=1034.564,-90.271,-80.249,168.020,39.410,157.361
C09959=1034.570,-90.022,-80.260,168.022,39.409,157.361
C09960=1034.576,-89.773,-80.271,168.025,39.408,157.361
C09961=1034.582,-89.522,-80.281,168.028,39.407,157.361
C09962=1034.588,-89.273,-80.291,168.031,39.407,157.361
C09963=1034.594,-89.023,-80.302,168.034,39.406,157.361
C09964=1034.601,-88.774,-80.312,168.036,39.405,157.361
C09965=1034.606,-88.524,-80.323,168.038,39.404,157.361
C09966=1034.612,-88.274,-80.334,168.041,39.403,157.361
C09967=1034.619,-88.024,-80.344,168.044,39.402,157.361
C09968=1034.625,-87.774,-80.354,168.046,39.401,157.361
C09969=1034.631,-87.525,-80.365,168.049,39.400,157.361
C09970=1034.637,-87.276,-80.376,168.052,39.400,157.361
C09971=1034.643,-87.025,-80.387,168.055,39.399,157.360
C09972=1034.649,-86.776,-80.396,168.058,39.398,157.360
C09973=1034.655,-86.526,-80.407,168.060,39.397,157.360
C09974=1034.662,-86.277,-80.417,168.063,39.396,157.360
C09975=1034.668,-86.027,-80.429,168.065,39.395,157.360
C09976=1034.674,-85.777,-80.440,168.068,39.394,157.360
C09977=1034.680,-85.527,-80.449,168.070,39.393,157.360
C09978=1034.686,-85.277,-80.460,168.073,39.393,157.360
C09979=1034.692,-85.028,-80.471,168.076,39.392,157.360
C09980=1034.698,-84.779,-80.482,168.079,39.391,157.360
C09981=1034.706,-84.493,-80.494,168.082,39.390,157.360
C09982=1034.712,-84.209,-80.506,168.085,39.389,157.360
C09983=1034.720,-83.923,-80.518,168.088,39.387,157.360
C09984=1034.727,-83.639,-80.530,168.091,39.387,157.360
C09985=1034.732,-83.389,-80.541,168.093,39.386,157.360
///RCONF 1,0,0,0,0,0,0,0,0,0,0,0,0,0,0,0,0,0,0,0,0,0,0,0
C09986=1034.739,-83.139,-80.552,168.096,39.385,157.359
C09987=1034.745,-82.890,-80.562,168.099,39.384,157.359
C09988=1034.751,-82.640,-80.573,168.101,39.383,157.359
C09989=1034.758,-82.390,-80.584,168.104,39.382,157.359
C09990=1034.764,-82.141,-80.595,168.107,39.381,157.359
C09991=1034.770,-81.891,-80.606,168.110,39.380,157.359
C09992=1034.776,-81.642,-80.616,168.112,39.380,157.359
C09993=1034.782,-81.392,-80.627,168.115,39.379,157.359
C09994=1034.789,-81.142,-80.638,168.118,39.379,157.359
C09995=1034.795,-80.893,-80.649,168.121,39.378,157.359
C09996=1034.801,-80.642,-80.660,168.123,39.377,157.359
//INST
///DATE 2021/06/17 10:57
///ATTR SC,RW,RJ
////FRAME ROBOT
///GROUP1 RB1
NOP
MOVL C00000 V=800.0 PL=0
MOVL C00001 V=800.0 PL=0
MOVL C00002 V=800.0 PL=0
MOVL C00003 V=800.0 PL=0
MOVL C00004 V=800.0 PL=0
MOVL C00005 V=800.0 PL=0
MOVL C00006 V=800.0 PL=0
MOVL C00007 V=800.0 PL=0
MOVL C00008 V=800.0 PL=0
MOVL C00009 V=800.0 PL=0
MOVL C00010 V=800.0 PL=0
MOVL C00011 V=800.0 PL=0
MOVL C00012 V=800.0 PL=0
MOVL C00013 V=800.0 PL=0
MOVL C00014 V=800.0 PL=0
MOVL C00015 V=800.0 PL=0
MOVL C00016 V=800.0 PL=0
MOVL C00017 V=800.0 PL=0
MOVL C00018 V=800.0 PL=0
MOVL C00019 V=800.0 PL=0
MOVL C00020 V=800.0 PL=0
MOVL C00021 V=800.0 PL=0
MOVL C00022 V=800.0 PL=0
MOVL C00023 V=800.0 PL=0
MOVL C00024 V=800.0 PL=0
MOVL C00025 V=800.0 PL=0
MOVL C00026 V=800.0 PL=0
MOVL C00027 V=800.0 PL=0
MOVL C00028 V=800.0 PL=0
MOVL C00029 V=800.0 PL=0
MOVL C00030 V=800.0 PL=0
MOVL C00031 V=800.0 PL=0
MOVL C00032 V=800.0 PL=0
MOVL C00033 V=800.0 PL=0
MOVL C00034 V=800.0 PL=0
MOVL C00035 V=800.0 PL=0
MOVL C00036 V=800.0 PL=0
MOVL C00037 V=800.0 PL=0
MOVL C00038 V=800.0 PL=0
MOVL C00039 V=800.0 PL=0
MOVL C00040 V=800.0 PL=0
MOVL C00041 V=800.0 PL=0
MOVL C00042 V=800.0 PL=0
MOVL C00043 V=800.0 PL=0
MOVL C00044 V=800.0 PL=0
MOVL C00045 V=800.0 PL=0
MOVL C00046 V=800.0 PL=0
MOVL C00047 V=800.0 PL=0
MOVL C00048 V=800.0 PL=0
MOVL C00049 V=800.0 PL=0
MOVL C00050 V=800.0 PL=0
MOVL C00051 V=800.0 PL=0
MOVL C00052 V=800.0 PL=0
MOVL C00053 V=800.0 PL=0
MOVL C00054 V=800.0 PL=0
MOVL C00055 V=800.0 PL=0
MOVL C00056 V=800.0 PL=0
MOVL C00057 V=800.0 PL=0
MOVL C00058 V=800.0 PL=0
MOVL C00059 V=800.0 PL=0
MOVL C00060 V=800.0 PL=0
MOVL C00061 V=800.0 PL=0
MOVL C00062 V=800.0 PL=0
MOVL C00063 V=800.0 PL=0
MOVL C00064 V=800.0 PL=0
MOVL C00065 V=800.0 PL=0
MOVL C00066 V=800.0 PL=0
MOVL C00067 V=800.0 PL=0
MOVL C00068 V=800.0 PL=0
MOVL C00069 V=800.0 PL=0
MOVL C00070 V=800.0 PL=0
MOVL C00071 V=800.0 PL=0
MOVL C00072 V=800.0 PL=0
MOVL C00073 V=800.0 PL=0
MOVL C00074 V=800.0 PL=0
MOVL C00075 V=800.0 PL=0
MOVL C00076 V=800.0 PL=0
MOVL C00077 V=800.0 PL=0
MOVL C00078 V=800.0 PL=0
MOVL C00079 V=800.0 PL=0
MOVL C00080 V=800.0 PL=0
MOVL C00081 V=800.0 PL=0
MOVL C00082 V=800.0 PL=0
MOVL C00083 V=800.0 PL=0
MOVL C00084 V=800.0 PL=0
MOVL C00085 V=800.0 PL=0
MOVL C00086 V=800.0 PL=0
MOVL C00087 V=800.0 PL=0
MOVL C00088 V=800.0 PL=0
MOVL C00089 V=800.0 PL=0
MOVL C00090 V=800.0 PL=0
MOVL C00091 V=800.0 PL=0
MOVL C00092 V=800.0 PL=0
MOVL C00093 V=800.0 PL=0
MOVL C00094 V=800.0 PL=0
MOVL C00095 V=800.0 PL=0
MOVL C00096 V=800.0 PL=0
MOVL C00097 V=800.0 PL=0
MOVL C00098 V=800.0 PL=0
MOVL C00099 V=800.0 PL=0
MOVL C00100 V=800.0 PL=0
MOVL C00101 V=800.0 PL=0
MOVL C00102 V=800.0 PL=0
MOVL C00103 V=800.0 PL=0
MOVL C00104 V=800.0 PL=0
MOVL C00105 V=800.0 PL=0
MOVL C00106 V=800.0 PL=0
MOVL C00107 V=800.0 PL=0
MOVL C00108 V=800.0 PL=0
MOVL C00109 V=800.0 PL=0
MOVL C00110 V=800.0 PL=0
MOVL C00111 V=800.0 PL=0
MOVL C00112 V=800.0 PL=0
MOVL C00113 V=800.0 PL=0
MOVL C00114 V=800.0 PL=0
MOVL C00115 V=800.0 PL=0
MOVL C00116 V=800.0 PL=0
MOVL C00117 V=800.0 PL=0
MOVL C00118 V=800.0 PL=0
MOVL C00119 V=800.0 PL=0
MOVL C00120 V=800.0 PL=0
MOVL C00121 V=800.0 PL=0
MOVL C00122 V=800.0 PL=0
MOVL C00123 V=800.0 PL=0
MOVL C00124 V=800.0 PL=0
MOVL C00125 V=800.0 PL=0
MOVL C00126 V=800.0 PL=0
MOVL C00127 V=800.0 PL=0
MOVL C00128 V=800.0 PL=0
MOVL C00129 V=800.0 PL=0
MOVL C00130 V=800.0 PL=0
MOVL C00131 V=800.0 PL=0
MOVL C00132 V=800.0 PL=0
MOVL C00133 V=800.0 PL=0
MOVL C00134 V=800.0 PL=0
MOVL C00135 V=800.0 PL=0
MOVL C00136 V=800.0 PL=0
MOVL C00137 V=800.0 PL=0
MOVL C00138 V=800.0 PL=0
MOVL C00139 V=800.0 PL=0
MOVL C00140 V=800.0 PL=0
MOVL C00141 V=800.0 PL=0
MOVL C00142 V=800.0 PL=0
MOVL C00143 V=800.0 PL=0
MOVL C00144 V=800.0 PL=0
MOVL C00145 V=800.0 PL=0
MOVL C00146 V=800.0 PL=0
MOVL C00147 V=800.0 PL=0
MOVL C00148 V=800.0 PL=0
MOVL C00149 V=800.0 PL=0
MOVL C00150 V=800.0 PL=0
MOVL C00151 V=800.0 PL=0
MOVL C00152 V=800.0 PL=0
MOVL C00153 V=800.0 PL=0
MOVL C00154 V=800.0 PL=0
MOVL C00155 V=800.0 PL=0
MOVL C00156 V=800.0 PL=0
MOVL C00157 V=800.0 PL=0
MOVL C00158 V=800.0 PL=0
MOVL C00159 V=800.0 PL=0
MOVL C00160 V=800.0 PL=0
MOVL C00161 V=800.0 PL=0
MOVL C00162 V=800.0 PL=0
MOVL C00163 V=800.0 PL=0
MOVL C00164 V=800.0 PL=0
MOVL C00165 V=800.0 PL=0
MOVL C00166 V=800.0 PL=0
MOVL C00167 V=800.0 PL=0
MOVL C00168 V=800.0 PL=0
MOVL C00169 V=800.0 PL=0
MOVL C00170 V=800.0 PL=0
MOVL C00171 V=800.0 PL=0
MOVL C00172 V=800.0 PL=0
MOVL C00173 V=800.0 PL=0
MOVL C00174 V=800.0 PL=0
MOVL C00175 V=800.0 PL=0
MOVL C00176 V=800.0 PL=0
MOVL C00177 V=800.0 PL=0
MOVL C00178 V=800.0 PL=0
MOVL C00179 V=800.0 PL=0
MOVL C00180 V=800.0 PL=0
MOVL C00181 V=800.0 PL=0
MOVL C00182 V=800.0 PL=0
MOVL C00183 V=800.0 PL=0
MOVL C00184 V=800.0 PL=0
MOVL C00185 V=800.0 PL=0
MOVL C00186 V=800.0 PL=0
MOVL C00187 V=800.0 PL=0
MOVL C00188 V=800.0 PL=0
MOVL C00189 V=800.0 PL=0
MOVL C00190 V=800.0 PL=0
MOVL C00191 V=800.0 PL=0
MOVL C00192 V=800.0 PL=0
MOVL C00193 V=800.0 PL=0
MOVL C00194 V=800.0 PL=0
MOVL C00195 V=800.0 PL=0
MOVL C00196 V=800.0 PL=0
MOVL C00197 V=800.0 PL=0
MOVL C00198 V=800.0 PL=0
MOVL C00199 V=800.0 PL=0
MOVL C00200 V=800.0 PL=0
MOVL C00201 V=800.0 PL=0
MOVL C00202 V=800.0 PL=0
MOVL C00203 V=800.0 PL=0
MOVL C00204 V=800.0 PL=0
MOVL C00205 V=800.0 PL=0
MOVL C00206 V=800.0 PL=0
MOVL C00207 V=800.0 PL=0
MOVL C00208 V=800.0 PL=0
MOVL C00209 V=800.0 PL=0
MOVL C00210 V=800.0 PL=0
MOVL C00211 V=800.0 PL=0
MOVL C00212 V=800.0 PL=0
MOVL C00213 V=800.0 PL=0
MOVL C00214 V=800.0 PL=0
MOVL C00215 V=800.0 PL=0
MOVL C00216 V=800.0 PL=0
MOVL C00217 V=800.0 PL=0
MOVL C00218 V=800.0 PL=0
MOVL C00219 V=800.0 PL=0
MOVL C00220 V=800.0 PL=0
MOVL C00221 V=800.0 PL=0
MOVL C00222 V=800.0 PL=0
MOVL C00223 V=800.0 PL=0
MOVL C00224 V=800.0 PL=0
MOVL C00225 V=800.0 PL=0
MOVL C00226 V=800.0 PL=0
MOVL C00227 V=800.0 PL=0
MOVL C00228 V=800.0 PL=0
MOVL C00229 V=800.0 PL=0
MOVL C00230 V=800.0 PL=0
MOVL C00231 V=800.0 PL=0
MOVL C00232 V=800.0 PL=0
MOVL C00233 V=800.0 PL=0
MOVL C00234 V=800.0 PL=0
MOVL C00235 V=800.0 PL=0
MOVL C00236 V=800.0 PL=0
MOVL C00237 V=800.0 PL=0
MOVL C00238 V=800.0 PL=0
MOVL C00239 V=800.0 PL=0
MOVL C00240 V=800.0 PL=0
MOVL C00241 V=800.0 PL=0
MOVL C00242 V=800.0 PL=0
MOVL C00243 V=800.0 PL=0
MOVL C00244 V=800.0 PL=0
MOVL C00245 V=800.0 PL=0
MOVL C00246 V=800.0 PL=0
MOVL C00247 V=800.0 PL=0
MOVL C00248 V=800.0 PL=0
MOVL C00249 V=800.0 PL=0
MOVL C00250 V=800.0 PL=0
MOVL C00251 V=800.0 PL=0
MOVL C00252 V=800.0 PL=0
MOVL C00253 V=800.0 PL=0
MOVL C00254 V=800.0 PL=0
MOVL C00255 V=800.0 PL=0
MOVL C00256 V=800.0 PL=0
MOVL C00257 V=800.0 PL=0
MOVL C00258 V=800.0 PL=0
MOVL C00259 V=800.0 PL=0
MOVL C00260 V=800.0 PL=0
MOVL C00261 V=800.0 PL=0
MOVL C00262 V=800.0 PL=0
MOVL C00263 V=800.0 PL=0
MOVL C00264 V=800.0 PL=0
MOVL C00265 V=800.0 PL=0
MOVL C00266 V=800.0 PL=0
MOVL C00267 V=800.0 PL=0
MOVL C00268 V=800.0 PL=0
MOVL C00269 V=800.0 PL=0
MOVL C00270 V=800.0 PL=0
MOVL C00271 V=800.0 PL=0
MOVL C00272 V=800.0 PL=0
MOVL C00273 V=800.0 PL=0
MOVL C00274 V=800.0 PL=0
MOVL C00275 V=800.0 PL=0
MOVL C00276 V=800.0 PL=0
MOVL C00277 V=800.0 PL=0
MOVL C00278 V=800.0 PL=0
MOVL C00279 V=800.0 PL=0
MOVL C00280 V=800.0 PL=0
MOVL C00281 V=800.0 PL=0
MOVL C00282 V=800.0 PL=0
MOVL C00283 V=800.0 PL=0
MOVL C00284 V=800.0 PL=0
MOVL C00285 V=800.0 PL=0
MOVL C00286 V=800.0 PL=0
MOVL C00287 V=800.0 PL=0
MOVL C00288 V=800.0 PL=0
MOVL C00289 V=800.0 PL=0
MOVL C00290 V=800.0 PL=0
MOVL C00291 V=800.0 PL=0
MOVL C00292 V=800.0 PL=0
MOVL C00293 V=800.0 PL=0
MOVL C00294 V=800.0 PL=0
MOVL C00295 V=800.0 PL=0
MOVL C00296 V=800.0 PL=0
MOVL C00297 V=800.0 PL=0
MOVL C00298 V=800.0 PL=0
MOVL C00299 V=800.0 PL=0
MOVL C00300 V=800.0 PL=0
MOVL C00301 V=800.0 PL=0
MOVL C00302 V=800.0 PL=0
MOVL C00303 V=800.0 PL=0
MOVL C00304 V=800.0 PL=0
MOVL C00305 V=800.0 PL=0
MOVL C00306 V=800.0 PL=0
MOVL C00307 V=800.0 PL=0
MOVL C00308 V=800.0 PL=0
MOVL C00309 V=800.0 PL=0
MOVL C00310 V=800.0 PL=0
MOVL C00311 V=800.0 PL=0
MOVL C00312 V=800.0 PL=0
MOVL C00313 V=800.0 PL=0
MOVL C00314 V=800.0 PL=0
MOVL C00315 V=800.0 PL=0
MOVL C00316 V=800.0 PL=0
MOVL C00317 V=800.0 PL=0
MOVL C00318 V=800.0 PL=0
MOVL C00319 V=800.0 PL=0
MOVL C00320 V=800.0 PL=0
MOVL C00321 V=800.0 PL=0
MOVL C00322 V=800.0 PL=0
MOVL C00323 V=800.0 PL=0
MOVL C00324 V=800.0 PL=0
MOVL C00325 V=800.0 PL=0
MOVL C00326 V=800.0 PL=0
MOVL C00327 V=800.0 PL=0
MOVL C00328 V=800.0 PL=0
MOVL C00329 V=800.0 PL=0
MOVL C00330 V=800.0 PL=0
MOVL C00331 V=800.0 PL=0
MOVL C00332 V=800.0 PL=0
MOVL C00333 V=800.0 PL=0
MOVL C00334 V=800.0 PL=0
MOVL C00335 V=800.0 PL=0
MOVL C00336 V=800.0 PL=0
MOVL C00337 V=800.0 PL=0
MOVL C00338 V=800.0 PL=0
MOVL C00339 V=800.0 PL=0
MOVL C00340 V=800.0 PL=0
MOVL C00341 V=800.0 PL=0
MOVL C00342 V=800.0 PL=0
MOVL C00343 V=800.0 PL=0
MOVL C00344 V=800.0 PL=0
MOVL C00345 V=800.0 PL=0
MOVL C00346 V=800.0 PL=0
MOVL C00347 V=800.0 PL=0
MOVL C00348 V=800.0 PL=0
MOVL C00349 V=800.0 PL=0
MOVL C00350 V=800.0 PL=0
MOVL C00351 V=800.0 PL=0
MOVL C00352 V=800.0 PL=0
MOVL C00353 V=800.0 PL=0
MOVL C00354 V=800.0 PL=0
MOVL C00355 V=800.0 PL=0
MOVL C00356 V=800.0 PL=0
MOVL C00357 V=800.0 PL=0
MOVL C00358 V=800.0 PL=0
MOVL C00359 V=800.0 PL=0
MOVL C00360 V=800.0 PL=0
MOVL C00361 V=800.0 PL=0
MOVL C00362 V=800.0 PL=0
MOVL C00363 V=800.0 PL=0
MOVL C00364 V=800.0 PL=0
MOVL C00365 V=800.0 PL=0
MOVL C00366 V=800.0 PL=0
MOVL C00367 V=800.0 PL=0
MOVL C00368 V=800.0 PL=0
MOVL C00369 V=800.0 PL=0
MOVL C00370 V=800.0 PL=0
MOVL C00371 V=800.0 PL=0
MOVL C00372 V=800.0 PL=0
MOVL C00373 V=800.0 PL=0
MOVL C00374 V=800.0 PL=0
MOVL C00375 V=800.0 PL=0
MOVL C00376 V=800.0 PL=0
MOVL C00377 V=800.0 PL=0
MOVL C00378 V=800.0 PL=0
MOVL C00379 V=800.0 PL=0
MOVL C00380 V=800.0 PL=0
MOVL C00381 V=800.0 PL=0
MOVL C00382 V=800.0 PL=0
MOVL C00383 V=800.0 PL=0
MOVL C00384 V=800.0 PL=0
MOVL C00385 V=800.0 PL=0
MOVL C00386 V=800.0 PL=0
MOVL C00387 V=800.0 PL=0
MOVL C00388 V=800.0 PL=0
MOVL C00389 V=800.0 PL=0
MOVL C00390 V=800.0 PL=0
MOVL C00391 V=800.0 PL=0
MOVL C00392 V=800.0 PL=0
MOVL C00393 V=800.0 PL=0
MOVL C00394 V=800.0 PL=0
MOVL C00395 V=800.0 PL=0
MOVL C00396 V=800.0 PL=0
MOVL C00397 V=800.0 PL=0
MOVL C00398 V=800.0 PL=0
MOVL C00399 V=800.0 PL=0
MOVL C00400 V=800.0 PL=0
MOVL C00401 V=800.0 PL=0
MOVL C00402 V=800.0 PL=0
MOVL C00403 V=800.0 PL=0
MOVL C00404 V=800.0 PL=0
MOVL C00405 V=800.0 PL=0
MOVL C00406 V=800.0 PL=0
MOVL C00407 V=800.0 PL=0
MOVL C00408 V=800.0 PL=0
MOVL C00409 V=800.0 PL=0
MOVL C00410 V=800.0 PL=0
MOVL C00411 V=800.0 PL=0
MOVL C00412 V=800.0 PL=0
MOVL C00413 V=800.0 PL=0
MOVL C00414 V=800.0 PL=0
MOVL C00415 V=800.0 PL=0
MOVL C00416 V=800.0 PL=0
MOVL C00417 V=800.0 PL=0
MOVL C00418 V=800.0 PL=0
MOVL C00419 V=800.0 PL=0
MOVL C00420 V=800.0 PL=0
MOVL C00421 V=800.0 PL=0
MOVL C00422 V=800.0 PL=0
MOVL C00423 V=800.0 PL=0
MOVL C00424 V=800.0 PL=0
MOVL C00425 V=800.0 PL=0
MOVL C00426 V=800.0 PL=0
MOVL C00427 V=800.0 PL=0
MOVL C00428 V=800.0 PL=0
MOVL C00429 V=800.0 PL=0
MOVL C00430 V=800.0 PL=0
MOVL C00431 V=800.0 PL=0
MOVL C00432 V=800.0 PL=0
MOVL C00433 V=800.0 PL=0
MOVL C00434 V=800.0 PL=0
MOVL C00435 V=800.0 PL=0
MOVL C00436 V=800.0 PL=0
MOVL C00437 V=800.0 PL=0
MOVL C00438 V=800.0 PL=0
MOVL C00439 V=800.0 PL=0
MOVL C00440 V=800.0 PL=0
MOVL C00441 V=800.0 PL=0
MOVL C00442 V=800.0 PL=0
MOVL C00443 V=800.0 PL=0
MOVL C00444 V=800.0 PL=0
MOVL C00445 V=800.0 PL=0
MOVL C00446 V=800.0 PL=0
MOVL C00447 V=800.0 PL=0
MOVL C00448 V=800.0 PL=0
MOVL C00449 V=800.0 PL=0
MOVL C00450 V=800.0 PL=0
MOVL C00451 V=800.0 PL=0
MOVL C00452 V=800.0 PL=0
MOVL C00453 V=800.0 PL=0
MOVL C00454 V=800.0 PL=0
MOVL C00455 V=800.0 PL=0
MOVL C00456 V=800.0 PL=0
MOVL C00457 V=800.0 PL=0
MOVL C00458 V=800.0 PL=0
MOVL C00459 V=800.0 PL=0
MOVL C00460 V=800.0 PL=0
MOVL C00461 V=800.0 PL=0
MOVL C00462 V=800.0 PL=0
MOVL C00463 V=800.0 PL=0
MOVL C00464 V=800.0 PL=0
MOVL C00465 V=800.0 PL=0
MOVL C00466 V=800.0 PL=0
MOVL C00467 V=800.0 PL=0
MOVL C00468 V=800.0 PL=0
MOVL C00469 V=800.0 PL=0
MOVL C00470 V=800.0 PL=0
MOVL C00471 V=800.0 PL=0
MOVL C00472 V=800.0 PL=0
MOVL C00473 V=800.0 PL=0
MOVL C00474 V=800.0 PL=0
MOVL C00475 V=800.0 PL=0
MOVL C00476 V=800.0 PL=0
MOVL C00477 V=800.0 PL=0
MOVL C00478 V=800.0 PL=0
MOVL C00479 V=800.0 PL=0
MOVL C00480 V=800.0 PL=0
MOVL C00481 V=800.0 PL=0
MOVL C00482 V=800.0 PL=0
MOVL C00483 V=800.0 PL=0
MOVL C00484 V=800.0 PL=0
MOVL C00485 V=800.0 PL=0
MOVL C00486 V=800.0 PL=0
MOVL C00487 V=800.0 PL=0
MOVL C00488 V=800.0 PL=0
MOVL C00489 V=800.0 PL=0
MOVL C00490 V=800.0 PL=0
MOVL C00491 V=800.0 PL=0
MOVL C00492 V=800.0 PL=0
MOVL C00493 V=800.0 PL=0
MOVL C00494 V=800.0 PL=0
MOVL C00495 V=800.0 PL=0
MOVL C00496 V=800.0 PL=0
MOVL C00497 V=800.0 PL=0
MOVL C00498 V=800.0 PL=0
MOVL C00499 V=800.0 PL=0
MOVL C00500 V=800.0 PL=0
MOVL C00501 V=800.0 PL=0
MOVL C00502 V=800.0 PL=0
MOVL C00503 V=800.0 PL=0
MOVL C00504 V=800.0 PL=0
MOVL C00505 V=800.0 PL=0
MOVL C00506 V=800.0 PL=0
MOVL C00507 V=800.0 PL=0
MOVL C00508 V=800.0 PL=0
MOVL C00509 V=800.0 PL=0
MOVL C00510 V=800.0 PL=0
MOVL C00511 V=800.0 PL=0
MOVL C00512 V=800.0 PL=0
MOVL C00513 V=800.0 PL=0
MOVL C00514 V=800.0 PL=0
MOVL C00515 V=800.0 PL=0
MOVL C00516 V=800.0 PL=0
MOVL C00517 V=800.0 PL=0
MOVL C00518 V=800.0 PL=0
MOVL C00519 V=800.0 PL=0
MOVL C00520 V=800.0 PL=0
MOVL C00521 V=800.0 PL=0
MOVL C00522 V=800.0 PL=0
MOVL C00523 V=800.0 PL=0
MOVL C00524 V=800.0 PL=0
MOVL C00525 V=800.0 PL=0
MOVL C00526 V=800.0 PL=0
MOVL C00527 V=800.0 PL=0
MOVL C00528 V=800.0 PL=0
MOVL C00529 V=800.0 PL=0
MOVL C00530 V=800.0 PL=0
MOVL C00531 V=800.0 PL=0
MOVL C00532 V=800.0 PL=0
MOVL C00533 V=800.0 PL=0
MOVL C00534 V=800.0 PL=0
MOVL C00535 V=800.0 PL=0
MOVL C00536 V=800.0 PL=0
MOVL C00537 V=800.0 PL=0
MOVL C00538 V=800.0 PL=0
MOVL C00539 V=800.0 PL=0
MOVL C00540 V=800.0 PL=0
MOVL C00541 V=800.0 PL=0
MOVL C00542 V=800.0 PL=0
MOVL C00543 V=800.0 PL=0
MOVL C00544 V=800.0 PL=0
MOVL C00545 V=800.0 PL=0
MOVL C00546 V=800.0 PL=0
MOVL C00547 V=800.0 PL=0
MOVL C00548 V=800.0 PL=0
MOVL C00549 V=800.0 PL=0
MOVL C00550 V=800.0 PL=0
MOVL C00551 V=800.0 PL=0
MOVL C00552 V=800.0 PL=0
MOVL C00553 V=800.0 PL=0
MOVL C00554 V=800.0 PL=0
MOVL C00555 V=800.0 PL=0
MOVL C00556 V=800.0 PL=0
MOVL C00557 V=800.0 PL=0
MOVL C00558 V=800.0 PL=0
MOVL C00559 V=800.0 PL=0
MOVL C00560 V=800.0 PL=0
MOVL C00561 V=800.0 PL=0
MOVL C00562 V=800.0 PL=0
MOVL C00563 V=800.0 PL=0
MOVL C00564 V=800.0 PL=0
MOVL C00565 V=800.0 PL=0
MOVL C00566 V=800.0 PL=0
MOVL C00567 V=800.0 PL=0
MOVL C00568 V=800.0 PL=0
MOVL C00569 V=800.0 PL=0
MOVL C00570 V=800.0 PL=0
MOVL C00571 V=800.0 PL=0
MOVL C00572 V=800.0 PL=0
MOVL C00573 V=800.0 PL=0
MOVL C00574 V=800.0 PL=0
MOVL C00575 V=800.0 PL=0
MOVL C00576 V=800.0 PL=0
MOVL C00577 V=800.0 PL=0
MOVL C00578 V=800.0 PL=0
MOVL C00579 V=800.0 PL=0
MOVL C00580 V=800.0 PL=0
MOVL C00581 V=800.0 PL=0
MOVL C00582 V=800.0 PL=0
MOVL C00583 V=800.0 PL=0
MOVL C00584 V=800.0 PL=0
MOVL C00585 V=800.0 PL=0
MOVL C00586 V=800.0 PL=0
MOVL C00587 V=800.0 PL=0
MOVL C00588 V=800.0 PL=0
MOVL C00589 V=800.0 PL=0
MOVL C00590 V=800.0 PL=0
MOVL C00591 V=800.0 PL=0
MOVL C00592 V=800.0 PL=0
MOVL C00593 V=800.0 PL=0
MOVL C00594 V=800.0 PL=0
MOVL C00595 V=800.0 PL=0
MOVL C00596 V=800.0 PL=0
MOVL C00597 V=800.0 PL=0
MOVL C00598 V=800.0 PL=0
MOVL C00599 V=800.0 PL=0
MOVL C00600 V=800.0 PL=0
MOVL C00601 V=800.0 PL=0
MOVL C00602 V=800.0 PL=0
MOVL C00603 V=800.0 PL=0
MOVL C00604 V=800.0 PL=0
MOVL C00605 V=800.0 PL=0
MOVL C00606 V=800.0 PL=0
MOVL C00607 V=800.0 PL=0
MOVL C00608 V=800.0 PL=0
MOVL C00609 V=800.0 PL=0
MOVL C00610 V=800.0 PL=0
MOVL C00611 V=800.0 PL=0
MOVL C00612 V=800.0 PL=0
MOVL C00613 V=800.0 PL=0
MOVL C00614 V=800.0 PL=0
MOVL C00615 V=800.0 PL=0
MOVL C00616 V=800.0 PL=0
MOVL C00617 V=800.0 PL=0
MOVL C00618 V=800.0 PL=0
MOVL C00619 V=800.0 PL=0
MOVL C00620 V=800.0 PL=0
MOVL C00621 V=800.0 PL=0
MOVL C00622 V=800.0 PL=0
MOVL C00623 V=800.0 PL=0
MOVL C00624 V=800.0 PL=0
MOVL C00625 V=800.0 PL=0
MOVL C00626 V=800.0 PL=0
MOVL C00627 V=800.0 PL=0
MOVL C00628 V=800.0 PL=0
MOVL C00629 V=800.0 PL=0
MOVL C00630 V=800.0 PL=0
MOVL C00631 V=800.0 PL=0
MOVL C00632 V=800.0 PL=0
MOVL C00633 V=800.0 PL=0
MOVL C00634 V=800.0 PL=0
MOVL C00635 V=800.0 PL=0
MOVL C00636 V=800.0 PL=0
MOVL C00637 V=800.0 PL=0
MOVL C00638 V=800.0 PL=0
MOVL C00639 V=800.0 PL=0
MOVL C00640 V=800.0 PL=0
MOVL C00641 V=800.0 PL=0
MOVL C00642 V=800.0 PL=0
MOVL C00643 V=800.0 PL=0
MOVL C00644 V=800.0 PL=0
MOVL C00645 V=800.0 PL=0
MOVL C00646 V=800.0 PL=0
MOVL C00647 V=800.0 PL=0
MOVL C00648 V=800.0 PL=0
MOVL C00649 V=800.0 PL=0
MOVL C00650 V=800.0 PL=0
MOVL C00651 V=800.0 PL=0
MOVL C00652 V=800.0 PL=0
MOVL C00653 V=800.0 PL=0
MOVL C00654 V=800.0 PL=0
MOVL C00655 V=800.0 PL=0
MOVL C00656 V=800.0 PL=0
MOVL C00657 V=800.0 PL=0
MOVL C00658 V=800.0 PL=0
MOVL C00659 V=800.0 PL=0
MOVL C00660 V=800.0 PL=0
MOVL C00661 V=800.0 PL=0
MOVL C00662 V=800.0 PL=0
MOVL C00663 V=800.0 PL=0
MOVL C00664 V=800.0 PL=0
MOVL C00665 V=800.0 PL=0
MOVL C00666 V=800.0 PL=0
MOVL C00667 V=800.0 PL=0
MOVL C00668 V=800.0 PL=0
MOVL C00669 V=800.0 PL=0
MOVL C00670 V=800.0 PL=0
MOVL C00671 V=800.0 PL=0
MOVL C00672 V=800.0 PL=0
MOVL C00673 V=800.0 PL=0
MOVL C00674 V=800.0 PL=0
MOVL C00675 V=800.0 PL=0
MOVL C00676 V=800.0 PL=0
MOVL C00677 V=800.0 PL=0
MOVL C00678 V=800.0 PL=0
MOVL C00679 V=800.0 PL=0
MOVL C00680 V=800.0 PL=0
MOVL C00681 V=800.0 PL=0
MOVL C00682 V=800.0 PL=0
MOVL C00683 V=800.0 PL=0
MOVL C00684 V=800.0 PL=0
MOVL C00685 V=800.0 PL=0
MOVL C00686 V=800.0 PL=0
MOVL C00687 V=800.0 PL=0
MOVL C00688 V=800.0 PL=0
MOVL C00689 V=800.0 PL=0
MOVL C00690 V=800.0 PL=0
MOVL C00691 V=800.0 PL=0
MOVL C00692 V=800.0 PL=0
MOVL C00693 V=800.0 PL=0
MOVL C00694 V=800.0 PL=0
MOVL C00695 V=800.0 PL=0
MOVL C00696 V=800.0 PL=0
MOVL C00697 V=800.0 PL=0
MOVL C00698 V=800.0 PL=0
MOVL C00699 V=800.0 PL=0
MOVL C00700 V=800.0 PL=0
MOVL C00701 V=800.0 PL=0
MOVL C00702 V=800.0 PL=0
MOVL C00703 V=800.0 PL=0
MOVL C00704 V=800.0 PL=0
MOVL C00705 V=800.0 PL=0
MOVL C00706 V=800.0 PL=0
MOVL C00707 V=800.0 PL=0
MOVL C00708 V=800.0 PL=0
MOVL C00709 V=800.0 PL=0
MOVL C00710 V=800.0 PL=0
MOVL C00711 V=800.0 PL=0
MOVL C00712 V=800.0 PL=0
MOVL C00713 V=800.0 PL=0
MOVL C00714 V=800.0 PL=0
MOVL C00715 V=800.0 PL=0
MOVL C00716 V=800.0 PL=0
MOVL C00717 V=800.0 PL=0
MOVL C00718 V=800.0 PL=0
MOVL C00719 V=800.0 PL=0
MOVL C00720 V=800.0 PL=0
MOVL C00721 V=800.0 PL=0
MOVL C00722 V=800.0 PL=0
MOVL C00723 V=800.0 PL=0
MOVL C00724 V=800.0 PL=0
MOVL C00725 V=800.0 PL=0
MOVL C00726 V=800.0 PL=0
MOVL C00727 V=800.0 PL=0
MOVL C00728 V=800.0 PL=0
MOVL C00729 V=800.0 PL=0
MOVL C00730 V=800.0 PL=0
MOVL C00731 V=800.0 PL=0
MOVL C00732 V=800.0 PL=0
MOVL C00733 V=800.0 PL=0
MOVL C00734 V=800.0 PL=0
MOVL C00735 V=800.0 PL=0
MOVL C00736 V=800.0 PL=0
MOVL C00737 V=800.0 PL=0
MOVL C00738 V=800.0 PL=0
MOVL C00739 V=800.0 PL=0
MOVL C00740 V=800.0 PL=0
MOVL C00741 V=800.0 PL=0
MOVL C00742 V=800.0 PL=0
MOVL C00743 V=800.0 PL=0
MOVL C00744 V=800.0 PL=0
MOVL C00745 V=800.0 PL=0
MOVL C00746 V=800.0 PL=0
MOVL C00747 V=800.0 PL=0
MOVL C00748 V=800.0 PL=0
MOVL C00749 V=800.0 PL=0
MOVL C00750 V=800.0 PL=0
MOVL C00751 V=800.0 PL=0
MOVL C00752 V=800.0 PL=0
MOVL C00753 V=800.0 PL=0
MOVL C00754 V=800.0 PL=0
MOVL C00755 V=800.0 PL=0
MOVL C00756 V=800.0 PL=0
MOVL C00757 V=800.0 PL=0
MOVL C00758 V=800.0 PL=0
MOVL C00759 V=800.0 PL=0
MOVL C00760 V=800.0 PL=0
MOVL C00761 V=800.0 PL=0
MOVL C00762 V=800.0 PL=0
MOVL C00763 V=800.0 PL=0
MOVL C00764 V=800.0 PL=0
MOVL C00765 V=800.0 PL=0
MOVL C00766 V=800.0 PL=0
MOVL C00767 V=800.0 PL=0
MOVL C00768 V=800.0 PL=0
MOVL C00769 V=800.0 PL=0
MOVL C00770 V=800.0 PL=0
MOVL C00771 V=800.0 PL=0
MOVL C00772 V=800.0 PL=0
MOVL C00773 V=800.0 PL=0
MOVL C00774 V=800.0 PL=0
MOVL C00775 V=800.0 PL=0
MOVL C00776 V=800.0 PL=0
MOVL C00777 V=800.0 PL=0
MOVL C00778 V=800.0 PL=0
MOVL C00779 V=800.0 PL=0
MOVL C00780 V=800.0 PL=0
MOVL C00781 V=800.0 PL=0
MOVL C00782 V=800.0 PL=0
MOVL C00783 V=800.0 PL=0
MOVL C00784 V=800.0 PL=0
MOVL C00785 V=800.0 PL=0
MOVL C00786 V=800.0 PL=0
MOVL C00787 V=800.0 PL=0
MOVL C00788 V=800.0 PL=0
MOVL C00789 V=800.0 PL=0
MOVL C00790 V=800.0 PL=0
MOVL C00791 V=800.0 PL=0
MOVL C00792 V=800.0 PL=0
MOVL C00793 V=800.0 PL=0
MOVL C00794 V=800.0 PL=0
MOVL C00795 V=800.0 PL=0
MOVL C00796 V=800.0 PL=0
MOVL C00797 V=800.0 PL=0
MOVL C00798 V=800.0 PL=0
MOVL C00799 V=800.0 PL=0
MOVL C00800 V=800.0 PL=0
MOVL C00801 V=800.0 PL=0
MOVL C00802 V=800.0 PL=0
MOVL C00803 V=800.0 PL=0
MOVL C00804 V=800.0 PL=0
MOVL C00805 V=800.0 PL=0
MOVL C00806 V=800.0 PL=0
MOVL C00807 V=800.0 PL=0
MOVL C00808 V=800.0 PL=0
MOVL C00809 V=800.0 PL=0
MOVL C00810 V=800.0 PL=0
MOVL C00811 V=800.0 PL=0
MOVL C00812 V=800.0 PL=0
MOVL C00813 V=800.0 PL=0
MOVL C00814 V=800.0 PL=0
MOVL C00815 V=800.0 PL=0
MOVL C00816 V=800.0 PL=0
MOVL C00817 V=800.0 PL=0
MOVL C00818 V=800.0 PL=0
MOVL C00819 V=800.0 PL=0
MOVL C00820 V=800.0 PL=0
MOVL C00821 V=800.0 PL=0
MOVL C00822 V=800.0 PL=0
MOVL C00823 V=800.0 PL=0
MOVL C00824 V=800.0 PL=0
MOVL C00825 V=800.0 PL=0
MOVL C00826 V=800.0 PL=0
MOVL C00827 V=800.0 PL=0
MOVL C00828 V=800.0 PL=0
MOVL C00829 V=800.0 PL=0
MOVL C00830 V=800.0 PL=0
MOVL C00831 V=800.0 PL=0
MOVL C00832 V=800.0 PL=0
MOVL C00833 V=800.0 PL=0
MOVL C00834 V=800.0 PL=0
MOVL C00835 V=800.0 PL=0
MOVL C00836 V=800.0 PL=0
MOVL C00837 V=800.0 PL=0
MOVL C00838 V=800.0 PL=0
MOVL C00839 V=800.0 PL=0
MOVL C00840 V=800.0 PL=0
MOVL C00841 V=800.0 PL=0
MOVL C00842 V=800.0 PL=0
MOVL C00843 V=800.0 PL=0
MOVL C00844 V=800.0 PL=0
MOVL C00845 V=800.0 PL=0
MOVL C00846 V=800.0 PL=0
MOVL C00847 V=800.0 PL=0
MOVL C00848 V=800.0 PL=0
MOVL C00849 V=800.0 PL=0
MOVL C00850 V=800.0 PL=0
MOVL C00851 V=800.0 PL=0
MOVL C00852 V=800.0 PL=0
MOVL C00853 V=800.0 PL=0
MOVL C00854 V=800.0 PL=0
MOVL C00855 V=800.0 PL=0
MOVL C00856 V=800.0 PL=0
MOVL C00857 V=800.0 PL=0
MOVL C00858 V=800.0 PL=0
MOVL C00859 V=800.0 PL=0
MOVL C00860 V=800.0 PL=0
MOVL C00861 V=800.0 PL=0
MOVL C00862 V=800.0 PL=0
MOVL C00863 V=800.0 PL=0
MOVL C00864 V=800.0 PL=0
MOVL C00865 V=800.0 PL=0
MOVL C00866 V=800.0 PL=0
MOVL C00867 V=800.0 PL=0
MOVL C00868 V=800.0 PL=0
MOVL C00869 V=800.0 PL=0
MOVL C00870 V=800.0 PL=0
MOVL C00871 V=800.0 PL=0
MOVL C00872 V=800.0 PL=0
MOVL C00873 V=800.0 PL=0
MOVL C00874 V=800.0 PL=0
MOVL C00875 V=800.0 PL=0
MOVL C00876 V=800.0 PL=0
MOVL C00877 V=800.0 PL=0
MOVL C00878 V=800.0 PL=0
MOVL C00879 V=800.0 PL=0
MOVL C00880 V=800.0 PL=0
MOVL C00881 V=800.0 PL=0
MOVL C00882 V=800.0 PL=0
MOVL C00883 V=800.0 PL=0
MOVL C00884 V=800.0 PL=0
MOVL C00885 V=800.0 PL=0
MOVL C00886 V=800.0 PL=0
MOVL C00887 V=800.0 PL=0
MOVL C00888 V=800.0 PL=0
MOVL C00889 V=800.0 PL=0
MOVL C00890 V=800.0 PL=0
MOVL C00891 V=800.0 PL=0
MOVL C00892 V=800.0 PL=0
MOVL C00893 V=800.0 PL=0
MOVL C00894 V=800.0 PL=0
MOVL C00895 V=800.0 PL=0
MOVL C00896 V=800.0 PL=0
MOVL C00897 V=800.0 PL=0
MOVL C00898 V=800.0 PL=0
MOVL C00899 V=800.0 PL=0
MOVL C00900 V=800.0 PL=0
MOVL C00901 V=800.0 PL=0
MOVL C00902 V=800.0 PL=0
MOVL C00903 V=800.0 PL=0
MOVL C00904 V=800.0 PL=0
MOVL C00905 V=800.0 PL=0
MOVL C00906 V=800.0 PL=0
MOVL C00907 V=800.0 PL=0
MOVL C00908 V=800.0 PL=0
MOVL C00909 V=800.0 PL=0
MOVL C00910 V=800.0 PL=0
MOVL C00911 V=800.0 PL=0
MOVL C00912 V=800.0 PL=0
MOVL C00913 V=800.0 PL=0
MOVL C00914 V=800.0 PL=0
MOVL C00915 V=800.0 PL=0
MOVL C00916 V=800.0 PL=0
MOVL C00917 V=800.0 PL=0
MOVL C00918 V=800.0 PL=0
MOVL C00919 V=800.0 PL=0
MOVL C00920 V=800.0 PL=0
MOVL C00921 V=800.0 PL=0
MOVL C00922 V=800.0 PL=0
MOVL C00923 V=800.0 PL=0
MOVL C00924 V=800.0 PL=0
MOVL C00925 V=800.0 PL=0
MOVL C00926 V=800.0 PL=0
MOVL C00927 V=800.0 PL=0
MOVL C00928 V=800.0 PL=0
MOVL C00929 V=800.0 PL=0
MOVL C00930 V=800.0 PL=0
MOVL C00931 V=800.0 PL=0
MOVL C00932 V=800.0 PL=0
MOVL C00933 V=800.0 PL=0
MOVL C00934 V=800.0 PL=0
MOVL C00935 V=800.0 PL=0
MOVL C00936 V=800.0 PL=0
MOVL C00937 V=800.0 PL=0
MOVL C00938 V=800.0 PL=0
MOVL C00939 V=800.0 PL=0
MOVL C00940 V=800.0 PL=0
MOVL C00941 V=800.0 PL=0
MOVL C00942 V=800.0 PL=0
MOVL C00943 V=800.0 PL=0
MOVL C00944 V=800.0 PL=0
MOVL C00945 V=800.0 PL=0
MOVL C00946 V=800.0 PL=0
MOVL C00947 V=800.0 PL=0
MOVL C00948 V=800.0 PL=0
MOVL C00949 V=800.0 PL=0
MOVL C00950 V=800.0 PL=0
MOVL C00951 V=800.0 PL=0
MOVL C00952 V=800.0 PL=0
MOVL C00953 V=800.0 PL=0
MOVL C00954 V=800.0 PL=0
MOVL C00955 V=800.0 PL=0
MOVL C00956 V=800.0 PL=0
MOVL C00957 V=800.0 PL=0
MOVL C00958 V=800.0 PL=0
MOVL C00959 V=800.0 PL=0
MOVL C00960 V=800.0 PL=0
MOVL C00961 V=800.0 PL=0
MOVL C00962 V=800.0 PL=0
MOVL C00963 V=800.0 PL=0
MOVL C00964 V=800.0 PL=0
MOVL C00965 V=800.0 PL=0
MOVL C00966 V=800.0 PL=0
MOVL C00967 V=800.0 PL=0
MOVL C00968 V=800.0 PL=0
MOVL C00969 V=800.0 PL=0
MOVL C00970 V=800.0 PL=0
MOVL C00971 V=800.0 PL=0
MOVL C00972 V=800.0 PL=0
MOVL C00973 V=800.0 PL=0
MOVL C00974 V=800.0 PL=0
MOVL C00975 V=800.0 PL=0
MOVL C00976 V=800.0 PL=0
MOVL C00977 V=800.0 PL=0
MOVL C00978 V=800.0 PL=0
MOVL C00979 V=800.0 PL=0
MOVL C00980 V=800.0 PL=0
MOVL C00981 V=800.0 PL=0
MOVL C00982 V=800.0 PL=0
MOVL C00983 V=800.0 PL=0
MOVL C00984 V=800.0 PL=0
MOVL C00985 V=800.0 PL=0
MOVL C00986 V=800.0 PL=0
MOVL C00987 V=800.0 PL=0
MOVL C00988 V=800.0 PL=0
MOVL C00989 V=800.0 PL=0
MOVL C00990 V=800.0 PL=0
MOVL C00991 V=800.0 PL=0
MOVL C00992 V=800.0 PL=0
MOVL C00993 V=800.0 PL=0
MOVL C00994 V=800.0 PL=0
MOVL C00995 V=800.0 PL=0
MOVL C00996 V=800.0 PL=0
MOVL C00997 V=800.0 PL=0
MOVL C00998 V=800.0 PL=0
MOVL C00999 V=800.0 PL=0
MOVL C01000 V=800.0 PL=0
MOVL C01001 V=800.0 PL=0
MOVL C01002 V=800.0 PL=0
MOVL C01003 V=800.0 PL=0
MOVL C01004 V=800.0 PL=0
MOVL C01005 V=800.0 PL=0
MOVL C01006 V=800.0 PL=0
MOVL C01007 V=800.0 PL=0
MOVL C01008 V=800.0 PL=0
MOVL C01009 V=800.0 PL=0
MOVL C01010 V=800.0 PL=0
MOVL C01011 V=800.0 PL=0
MOVL C01012 V=800.0 PL=0
MOVL C01013 V=800.0 PL=0
MOVL C01014 V=800.0 PL=0
MOVL C01015 V=800.0 PL=0
MOVL C01016 V=800.0 PL=0
MOVL C01017 V=800.0 PL=0
MOVL C01018 V=800.0 PL=0
MOVL C01019 V=800.0 PL=0
MOVL C01020 V=800.0 PL=0
MOVL C01021 V=800.0 PL=0
MOVL C01022 V=800.0 PL=0
MOVL C01023 V=800.0 PL=0
MOVL C01024 V=800.0 PL=0
MOVL C01025 V=800.0 PL=0
MOVL C01026 V=800.0 PL=0
MOVL C01027 V=800.0 PL=0
MOVL C01028 V=800.0 PL=0
MOVL C01029 V=800.0 PL=0
MOVL C01030 V=800.0 PL=0
MOVL C01031 V=800.0 PL=0
MOVL C01032 V=800.0 PL=0
MOVL C01033 V=800.0 PL=0
MOVL C01034 V=800.0 PL=0
MOVL C01035 V=800.0 PL=0
MOVL C01036 V=800.0 PL=0
MOVL C01037 V=800.0 PL=0
MOVL C01038 V=800.0 PL=0
MOVL C01039 V=800.0 PL=0
MOVL C01040 V=800.0 PL=0
MOVL C01041 V=800.0 PL=0
MOVL C01042 V=800.0 PL=0
MOVL C01043 V=800.0 PL=0
MOVL C01044 V=800.0 PL=0
MOVL C01045 V=800.0 PL=0
MOVL C01046 V=800.0 PL=0
MOVL C01047 V=800.0 PL=0
MOVL C01048 V=800.0 PL=0
MOVL C01049 V=800.0 PL=0
MOVL C01050 V=800.0 PL=0
MOVL C01051 V=800.0 PL=0
MOVL C01052 V=800.0 PL=0
MOVL C01053 V=800.0 PL=0
MOVL C01054 V=800.0 PL=0
MOVL C01055 V=800.0 PL=0
MOVL C01056 V=800.0 PL=0
MOVL C01057 V=800.0 PL=0
MOVL C01058 V=800.0 PL=0
MOVL C01059 V=800.0 PL=0
MOVL C01060 V=800.0 PL=0
MOVL C01061 V=800.0 PL=0
MOVL C01062 V=800.0 PL=0
MOVL C01063 V=800.0 PL=0
MOVL C01064 V=800.0 PL=0
MOVL C01065 V=800.0 PL=0
MOVL C01066 V=800.0 PL=0
MOVL C01067 V=800.0 PL=0
MOVL C01068 V=800.0 PL=0
MOVL C01069 V=800.0 PL=0
MOVL C01070 V=800.0 PL=0
MOVL C01071 V=800.0 PL=0
MOVL C01072 V=800.0 PL=0
MOVL C01073 V=800.0 PL=0
MOVL C01074 V=800.0 PL=0
MOVL C01075 V=800.0 PL=0
MOVL C01076 V=800.0 PL=0
MOVL C01077 V=800.0 PL=0
MOVL C01078 V=800.0 PL=0
MOVL C01079 V=800.0 PL=0
MOVL C01080 V=800.0 PL=0
MOVL C01081 V=800.0 PL=0
MOVL C01082 V=800.0 PL=0
MOVL C01083 V=800.0 PL=0
MOVL C01084 V=800.0 PL=0
MOVL C01085 V=800.0 PL=0
MOVL C01086 V=800.0 PL=0
MOVL C01087 V=800.0 PL=0
MOVL C01088 V=800.0 PL=0
MOVL C01089 V=800.0 PL=0
MOVL C01090 V=800.0 PL=0
MOVL C01091 V=800.0 PL=0
MOVL C01092 V=800.0 PL=0
MOVL C01093 V=800.0 PL=0
MOVL C01094 V=800.0 PL=0
MOVL C01095 V=800.0 PL=0
MOVL C01096 V=800.0 PL=0
MOVL C01097 V=800.0 PL=0
MOVL C01098 V=800.0 PL=0
MOVL C01099 V=800.0 PL=0
MOVL C01100 V=800.0 PL=0
MOVL C01101 V=800.0 PL=0
MOVL C01102 V=800.0 PL=0
MOVL C01103 V=800.0 PL=0
MOVL C01104 V=800.0 PL=0
MOVL C01105 V=800.0 PL=0
MOVL C01106 V=800.0 PL=0
MOVL C01107 V=800.0 PL=0
MOVL C01108 V=800.0 PL=0
MOVL C01109 V=800.0 PL=0
MOVL C01110 V=800.0 PL=0
MOVL C01111 V=800.0 PL=0
MOVL C01112 V=800.0 PL=0
MOVL C01113 V=800.0 PL=0
MOVL C01114 V=800.0 PL=0
MOVL C01115 V=800.0 PL=0
MOVL C01116 V=800.0 PL=0
MOVL C01117 V=800.0 PL=0
MOVL C01118 V=800.0 PL=0
MOVL C01119 V=800.0 PL=0
MOVL C01120 V=800.0 PL=0
MOVL C01121 V=800.0 PL=0
MOVL C01122 V=800.0 PL=0
MOVL C01123 V=800.0 PL=0
MOVL C01124 V=800.0 PL=0
MOVL C01125 V=800.0 PL=0
MOVL C01126 V=800.0 PL=0
MOVL C01127 V=800.0 PL=0
MOVL C01128 V=800.0 PL=0
MOVL C01129 V=800.0 PL=0
MOVL C01130 V=800.0 PL=0
MOVL C01131 V=800.0 PL=0
MOVL C01132 V=800.0 PL=0
MOVL C01133 V=800.0 PL=0
MOVL C01134 V=800.0 PL=0
MOVL C01135 V=800.0 PL=0
MOVL C01136 V=800.0 PL=0
MOVL C01137 V=800.0 PL=0
MOVL C01138 V=800.0 PL=0
MOVL C01139 V=800.0 PL=0
MOVL C01140 V=800.0 PL=0
MOVL C01141 V=800.0 PL=0
MOVL C01142 V=800.0 PL=0
MOVL C01143 V=800.0 PL=0
MOVL C01144 V=800.0 PL=0
MOVL C01145 V=800.0 PL=0
MOVL C01146 V=800.0 PL=0
MOVL C01147 V=800.0 PL=0
MOVL C01148 V=800.0 PL=0
MOVL C01149 V=800.0 PL=0
MOVL C01150 V=800.0 PL=0
MOVL C01151 V=800.0 PL=0
MOVL C01152 V=800.0 PL=0
MOVL C01153 V=800.0 PL=0
MOVL C01154 V=800.0 PL=0
MOVL C01155 V=800.0 PL=0
MOVL C01156 V=800.0 PL=0
MOVL C01157 V=800.0 PL=0
MOVL C01158 V=800.0 PL=0
MOVL C01159 V=800.0 PL=0
MOVL C01160 V=800.0 PL=0
MOVL C01161 V=800.0 PL=0
MOVL C01162 V=800.0 PL=0
MOVL C01163 V=800.0 PL=0
MOVL C01164 V=800.0 PL=0
MOVL C01165 V=800.0 PL=0
MOVL C01166 V=800.0 PL=0
MOVL C01167 V=800.0 PL=0
MOVL C01168 V=800.0 PL=0
MOVL C01169 V=800.0 PL=0
MOVL C01170 V=800.0 PL=0
MOVL C01171 V=800.0 PL=0
MOVL C01172 V=800.0 PL=0
MOVL C01173 V=800.0 PL=0
MOVL C01174 V=800.0 PL=0
MOVL C01175 V=800.0 PL=0
MOVL C01176 V=800.0 PL=0
MOVL C01177 V=800.0 PL=0
MOVL C01178 V=800.0 PL=0
MOVL C01179 V=800.0 PL=0
MOVL C01180 V=800.0 PL=0
MOVL C01181 V=800.0 PL=0
MOVL C01182 V=800.0 PL=0
MOVL C01183 V=800.0 PL=0
MOVL C01184 V=800.0 PL=0
MOVL C01185 V=800.0 PL=0
MOVL C01186 V=800.0 PL=0
MOVL C01187 V=800.0 PL=0
MOVL C01188 V=800.0 PL=0
MOVL C01189 V=800.0 PL=0
MOVL C01190 V=800.0 PL=0
MOVL C01191 V=800.0 PL=0
MOVL C01192 V=800.0 PL=0
MOVL C01193 V=800.0 PL=0
MOVL C01194 V=800.0 PL=0
MOVL C01195 V=800.0 PL=0
MOVL C01196 V=800.0 PL=0
MOVL C01197 V=800.0 PL=0
MOVL C01198 V=800.0 PL=0
MOVL C01199 V=800.0 PL=0
MOVL C01200 V=800.0 PL=0
MOVL C01201 V=800.0 PL=0
MOVL C01202 V=800.0 PL=0
MOVL C01203 V=800.0 PL=0
MOVL C01204 V=800.0 PL=0
MOVL C01205 V=800.0 PL=0
MOVL C01206 V=800.0 PL=0
MOVL C01207 V=800.0 PL=0
MOVL C01208 V=800.0 PL=0
MOVL C01209 V=800.0 PL=0
MOVL C01210 V=800.0 PL=0
MOVL C01211 V=800.0 PL=0
MOVL C01212 V=800.0 PL=0
MOVL C01213 V=800.0 PL=0
MOVL C01214 V=800.0 PL=0
MOVL C01215 V=800.0 PL=0
MOVL C01216 V=800.0 PL=0
MOVL C01217 V=800.0 PL=0
MOVL C01218 V=800.0 PL=0
MOVL C01219 V=800.0 PL=0
MOVL C01220 V=800.0 PL=0
MOVL C01221 V=800.0 PL=0
MOVL C01222 V=800.0 PL=0
MOVL C01223 V=800.0 PL=0
MOVL C01224 V=800.0 PL=0
MOVL C01225 V=800.0 PL=0
MOVL C01226 V=800.0 PL=0
MOVL C01227 V=800.0 PL=0
MOVL C01228 V=800.0 PL=0
MOVL C01229 V=800.0 PL=0
MOVL C01230 V=800.0 PL=0
MOVL C01231 V=800.0 PL=0
MOVL C01232 V=800.0 PL=0
MOVL C01233 V=800.0 PL=0
MOVL C01234 V=800.0 PL=0
MOVL C01235 V=800.0 PL=0
MOVL C01236 V=800.0 PL=0
MOVL C01237 V=800.0 PL=0
MOVL C01238 V=800.0 PL=0
MOVL C01239 V=800.0 PL=0
MOVL C01240 V=800.0 PL=0
MOVL C01241 V=800.0 PL=0
MOVL C01242 V=800.0 PL=0
MOVL C01243 V=800.0 PL=0
MOVL C01244 V=800.0 PL=0
MOVL C01245 V=800.0 PL=0
MOVL C01246 V=800.0 PL=0
MOVL C01247 V=800.0 PL=0
MOVL C01248 V=800.0 PL=0
MOVL C01249 V=800.0 PL=0
MOVL C01250 V=800.0 PL=0
MOVL C01251 V=800.0 PL=0
MOVL C01252 V=800.0 PL=0
MOVL C01253 V=800.0 PL=0
MOVL C01254 V=800.0 PL=0
MOVL C01255 V=800.0 PL=0
MOVL C01256 V=800.0 PL=0
MOVL C01257 V=800.0 PL=0
MOVL C01258 V=800.0 PL=0
MOVL C01259 V=800.0 PL=0
MOVL C01260 V=800.0 PL=0
MOVL C01261 V=800.0 PL=0
MOVL C01262 V=800.0 PL=0
MOVL C01263 V=800.0 PL=0
MOVL C01264 V=800.0 PL=0
MOVL C01265 V=800.0 PL=0
MOVL C01266 V=800.0 PL=0
MOVL C01267 V=800.0 PL=0
MOVL C01268 V=800.0 PL=0
MOVL C01269 V=800.0 PL=0
MOVL C01270 V=800.0 PL=0
MOVL C01271 V=800.0 PL=0
MOVL C01272 V=800.0 PL=0
MOVL C01273 V=800.0 PL=0
MOVL C01274 V=800.0 PL=0
MOVL C01275 V=800.0 PL=0
MOVL C01276 V=800.0 PL=0
MOVL C01277 V=800.0 PL=0
MOVL C01278 V=800.0 PL=0
MOVL C01279 V=800.0 PL=0
MOVL C01280 V=800.0 PL=0
MOVL C01281 V=800.0 PL=0
MOVL C01282 V=800.0 PL=0
MOVL C01283 V=800.0 PL=0
MOVL C01284 V=800.0 PL=0
MOVL C01285 V=800.0 PL=0
MOVL C01286 V=800.0 PL=0
MOVL C01287 V=800.0 PL=0
MOVL C01288 V=800.0 PL=0
MOVL C01289 V=800.0 PL=0
MOVL C01290 V=800.0 PL=0
MOVL C01291 V=800.0 PL=0
MOVL C01292 V=800.0 PL=0
MOVL C01293 V=800.0 PL=0
MOVL C01294 V=800.0 PL=0
MOVL C01295 V=800.0 PL=0
MOVL C01296 V=800.0 PL=0
MOVL C01297 V=800.0 PL=0
MOVL C01298 V=800.0 PL=0
MOVL C01299 V=800.0 PL=0
MOVL C01300 V=800.0 PL=0
MOVL C01301 V=800.0 PL=0
MOVL C01302 V=800.0 PL=0
MOVL C01303 V=800.0 PL=0
MOVL C01304 V=800.0 PL=0
MOVL C01305 V=800.0 PL=0
MOVL C01306 V=800.0 PL=0
MOVL C01307 V=800.0 PL=0
MOVL C01308 V=800.0 PL=0
MOVL C01309 V=800.0 PL=0
MOVL C01310 V=800.0 PL=0
MOVL C01311 V=800.0 PL=0
MOVL C01312 V=800.0 PL=0
MOVL C01313 V=800.0 PL=0
MOVL C01314 V=800.0 PL=0
MOVL C01315 V=800.0 PL=0
MOVL C01316 V=800.0 PL=0
MOVL C01317 V=800.0 PL=0
MOVL C01318 V=800.0 PL=0
MOVL C01319 V=800.0 PL=0
MOVL C01320 V=800.0 PL=0
MOVL C01321 V=800.0 PL=0
MOVL C01322 V=800.0 PL=0
MOVL C01323 V=800.0 PL=0
MOVL C01324 V=800.0 PL=0
MOVL C01325 V=800.0 PL=0
MOVL C01326 V=800.0 PL=0
MOVL C01327 V=800.0 PL=0
MOVL C01328 V=800.0 PL=0
MOVL C01329 V=800.0 PL=0
MOVL C01330 V=800.0 PL=0
MOVL C01331 V=800.0 PL=0
MOVL C01332 V=800.0 PL=0
MOVL C01333 V=800.0 PL=0
MOVL C01334 V=800.0 PL=0
MOVL C01335 V=800.0 PL=0
MOVL C01336 V=800.0 PL=0
MOVL C01337 V=800.0 PL=0
MOVL C01338 V=800.0 PL=0
MOVL C01339 V=800.0 PL=0
MOVL C01340 V=800.0 PL=0
MOVL C01341 V=800.0 PL=0
MOVL C01342 V=800.0 PL=0
MOVL C01343 V=800.0 PL=0
MOVL C01344 V=800.0 PL=0
MOVL C01345 V=800.0 PL=0
MOVL C01346 V=800.0 PL=0
MOVL C01347 V=800.0 PL=0
MOVL C01348 V=800.0 PL=0
MOVL C01349 V=800.0 PL=0
MOVL C01350 V=800.0 PL=0
MOVL C01351 V=800.0 PL=0
MOVL C01352 V=800.0 PL=0
MOVL C01353 V=800.0 PL=0
MOVL C01354 V=800.0 PL=0
MOVL C01355 V=800.0 PL=0
MOVL C01356 V=800.0 PL=0
MOVL C01357 V=800.0 PL=0
MOVL C01358 V=800.0 PL=0
MOVL C01359 V=800.0 PL=0
MOVL C01360 V=800.0 PL=0
MOVL C01361 V=800.0 PL=0
MOVL C01362 V=800.0 PL=0
MOVL C01363 V=800.0 PL=0
MOVL C01364 V=800.0 PL=0
MOVL C01365 V=800.0 PL=0
MOVL C01366 V=800.0 PL=0
MOVL C01367 V=800.0 PL=0
MOVL C01368 V=800.0 PL=0
MOVL C01369 V=800.0 PL=0
MOVL C01370 V=800.0 PL=0
MOVL C01371 V=800.0 PL=0
MOVL C01372 V=800.0 PL=0
MOVL C01373 V=800.0 PL=0
MOVL C01374 V=800.0 PL=0
MOVL C01375 V=800.0 PL=0
MOVL C01376 V=800.0 PL=0
MOVL C01377 V=800.0 PL=0
MOVL C01378 V=800.0 PL=0
MOVL C01379 V=800.0 PL=0
MOVL C01380 V=800.0 PL=0
MOVL C01381 V=800.0 PL=0
MOVL C01382 V=800.0 PL=0
MOVL C01383 V=800.0 PL=0
MOVL C01384 V=800.0 PL=0
MOVL C01385 V=800.0 PL=0
MOVL C01386 V=800.0 PL=0
MOVL C01387 V=800.0 PL=0
MOVL C01388 V=800.0 PL=0
MOVL C01389 V=800.0 PL=0
MOVL C01390 V=800.0 PL=0
MOVL C01391 V=800.0 PL=0
MOVL C01392 V=800.0 PL=0
MOVL C01393 V=800.0 PL=0
MOVL C01394 V=800.0 PL=0
MOVL C01395 V=800.0 PL=0
MOVL C01396 V=800.0 PL=0
MOVL C01397 V=800.0 PL=0
MOVL C01398 V=800.0 PL=0
MOVL C01399 V=800.0 PL=0
MOVL C01400 V=800.0 PL=0
MOVL C01401 V=800.0 PL=0
MOVL C01402 V=800.0 PL=0
MOVL C01403 V=800.0 PL=0
MOVL C01404 V=800.0 PL=0
MOVL C01405 V=800.0 PL=0
MOVL C01406 V=800.0 PL=0
MOVL C01407 V=800.0 PL=0
MOVL C01408 V=800.0 PL=0
MOVL C01409 V=800.0 PL=0
MOVL C01410 V=800.0 PL=0
MOVL C01411 V=800.0 PL=0
MOVL C01412 V=800.0 PL=0
MOVL C01413 V=800.0 PL=0
MOVL C01414 V=800.0 PL=0
MOVL C01415 V=800.0 PL=0
MOVL C01416 V=800.0 PL=0
MOVL C01417 V=800.0 PL=0
MOVL C01418 V=800.0 PL=0
MOVL C01419 V=800.0 PL=0
MOVL C01420 V=800.0 PL=0
MOVL C01421 V=800.0 PL=0
MOVL C01422 V=800.0 PL=0
MOVL C01423 V=800.0 PL=0
MOVL C01424 V=800.0 PL=0
MOVL C01425 V=800.0 PL=0
MOVL C01426 V=800.0 PL=0
MOVL C01427 V=800.0 PL=0
MOVL C01428 V=800.0 PL=0
MOVL C01429 V=800.0 PL=0
MOVL C01430 V=800.0 PL=0
MOVL C01431 V=800.0 PL=0
MOVL C01432 V=800.0 PL=0
MOVL C01433 V=800.0 PL=0
MOVL C01434 V=800.0 PL=0
MOVL C01435 V=800.0 PL=0
MOVL C01436 V=800.0 PL=0
MOVL C01437 V=800.0 PL=0
MOVL C01438 V=800.0 PL=0
MOVL C01439 V=800.0 PL=0
MOVL C01440 V=800.0 PL=0
MOVL C01441 V=800.0 PL=0
MOVL C01442 V=800.0 PL=0
MOVL C01443 V=800.0 PL=0
MOVL C01444 V=800.0 PL=0
MOVL C01445 V=800.0 PL=0
MOVL C01446 V=800.0 PL=0
MOVL C01447 V=800.0 PL=0
MOVL C01448 V=800.0 PL=0
MOVL C01449 V=800.0 PL=0
MOVL C01450 V=800.0 PL=0
MOVL C01451 V=800.0 PL=0
MOVL C01452 V=800.0 PL=0
MOVL C01453 V=800.0 PL=0
MOVL C01454 V=800.0 PL=0
MOVL C01455 V=800.0 PL=0
MOVL C01456 V=800.0 PL=0
MOVL C01457 V=800.0 PL=0
MOVL C01458 V=800.0 PL=0
MOVL C01459 V=800.0 PL=0
MOVL C01460 V=800.0 PL=0
MOVL C01461 V=800.0 PL=0
MOVL C01462 V=800.0 PL=0
MOVL C01463 V=800.0 PL=0
MOVL C01464 V=800.0 PL=0
MOVL C01465 V=800.0 PL=0
MOVL C01466 V=800.0 PL=0
MOVL C01467 V=800.0 PL=0
MOVL C01468 V=800.0 PL=0
MOVL C01469 V=800.0 PL=0
MOVL C01470 V=800.0 PL=0
MOVL C01471 V=800.0 PL=0
MOVL C01472 V=800.0 PL=0
MOVL C01473 V=800.0 PL=0
MOVL C01474 V=800.0 PL=0
MOVL C01475 V=800.0 PL=0
MOVL C01476 V=800.0 PL=0
MOVL C01477 V=800.0 PL=0
MOVL C01478 V=800.0 PL=0
MOVL C01479 V=800.0 PL=0
MOVL C01480 V=800.0 PL=0
MOVL C01481 V=800.0 PL=0
MOVL C01482 V=800.0 PL=0
MOVL C01483 V=800.0 PL=0
MOVL C01484 V=800.0 PL=0
MOVL C01485 V=800.0 PL=0
MOVL C01486 V=800.0 PL=0
MOVL C01487 V=800.0 PL=0
MOVL C01488 V=800.0 PL=0
MOVL C01489 V=800.0 PL=0
MOVL C01490 V=800.0 PL=0
MOVL C01491 V=800.0 PL=0
MOVL C01492 V=800.0 PL=0
MOVL C01493 V=800.0 PL=0
MOVL C01494 V=800.0 PL=0
MOVL C01495 V=800.0 PL=0
MOVL C01496 V=800.0 PL=0
MOVL C01497 V=800.0 PL=0
MOVL C01498 V=800.0 PL=0
MOVL C01499 V=800.0 PL=0
MOVL C01500 V=800.0 PL=0
MOVL C01501 V=800.0 PL=0
MOVL C01502 V=800.0 PL=0
MOVL C01503 V=800.0 PL=0
MOVL C01504 V=800.0 PL=0
MOVL C01505 V=800.0 PL=0
MOVL C01506 V=800.0 PL=0
MOVL C01507 V=800.0 PL=0
MOVL C01508 V=800.0 PL=0
MOVL C01509 V=800.0 PL=0
MOVL C01510 V=800.0 PL=0
MOVL C01511 V=800.0 PL=0
MOVL C01512 V=800.0 PL=0
MOVL C01513 V=800.0 PL=0
MOVL C01514 V=800.0 PL=0
MOVL C01515 V=800.0 PL=0
MOVL C01516 V=800.0 PL=0
MOVL C01517 V=800.0 PL=0
MOVL C01518 V=800.0 PL=0
MOVL C01519 V=800.0 PL=0
MOVL C01520 V=800.0 PL=0
MOVL C01521 V=800.0 PL=0
MOVL C01522 V=800.0 PL=0
MOVL C01523 V=800.0 PL=0
MOVL C01524 V=800.0 PL=0
MOVL C01525 V=800.0 PL=0
MOVL C01526 V=800.0 PL=0
MOVL C01527 V=800.0 PL=0
MOVL C01528 V=800.0 PL=0
MOVL C01529 V=800.0 PL=0
MOVL C01530 V=800.0 PL=0
MOVL C01531 V=800.0 PL=0
MOVL C01532 V=800.0 PL=0
MOVL C01533 V=800.0 PL=0
MOVL C01534 V=800.0 PL=0
MOVL C01535 V=800.0 PL=0
MOVL C01536 V=800.0 PL=0
MOVL C01537 V=800.0 PL=0
MOVL C01538 V=800.0 PL=0
MOVL C01539 V=800.0 PL=0
MOVL C01540 V=800.0 PL=0
MOVL C01541 V=800.0 PL=0
MOVL C01542 V=800.0 PL=0
MOVL C01543 V=800.0 PL=0
MOVL C01544 V=800.0 PL=0
MOVL C01545 V=800.0 PL=0
MOVL C01546 V=800.0 PL=0
MOVL C01547 V=800.0 PL=0
MOVL C01548 V=800.0 PL=0
MOVL C01549 V=800.0 PL=0
MOVL C01550 V=800.0 PL=0
MOVL C01551 V=800.0 PL=0
MOVL C01552 V=800.0 PL=0
MOVL C01553 V=800.0 PL=0
MOVL C01554 V=800.0 PL=0
MOVL C01555 V=800.0 PL=0
MOVL C01556 V=800.0 PL=0
MOVL C01557 V=800.0 PL=0
MOVL C01558 V=800.0 PL=0
MOVL C01559 V=800.0 PL=0
MOVL C01560 V=800.0 PL=0
MOVL C01561 V=800.0 PL=0
MOVL C01562 V=800.0 PL=0
MOVL C01563 V=800.0 PL=0
MOVL C01564 V=800.0 PL=0
MOVL C01565 V=800.0 PL=0
MOVL C01566 V=800.0 PL=0
MOVL C01567 V=800.0 PL=0
MOVL C01568 V=800.0 PL=0
MOVL C01569 V=800.0 PL=0
MOVL C01570 V=800.0 PL=0
MOVL C01571 V=800.0 PL=0
MOVL C01572 V=800.0 PL=0
MOVL C01573 V=800.0 PL=0
MOVL C01574 V=800.0 PL=0
MOVL C01575 V=800.0 PL=0
MOVL C01576 V=800.0 PL=0
MOVL C01577 V=800.0 PL=0
MOVL C01578 V=800.0 PL=0
MOVL C01579 V=800.0 PL=0
MOVL C01580 V=800.0 PL=0
MOVL C01581 V=800.0 PL=0
MOVL C01582 V=800.0 PL=0
MOVL C01583 V=800.0 PL=0
MOVL C01584 V=800.0 PL=0
MOVL C01585 V=800.0 PL=0
MOVL C01586 V=800.0 PL=0
MOVL C01587 V=800.0 PL=0
MOVL C01588 V=800.0 PL=0
MOVL C01589 V=800.0 PL=0
MOVL C01590 V=800.0 PL=0
MOVL C01591 V=800.0 PL=0
MOVL C01592 V=800.0 PL=0
MOVL C01593 V=800.0 PL=0
MOVL C01594 V=800.0 PL=0
MOVL C01595 V=800.0 PL=0
MOVL C01596 V=800.0 PL=0
MOVL C01597 V=800.0 PL=0
MOVL C01598 V=800.0 PL=0
MOVL C01599 V=800.0 PL=0
MOVL C01600 V=800.0 PL=0
MOVL C01601 V=800.0 PL=0
MOVL C01602 V=800.0 PL=0
MOVL C01603 V=800.0 PL=0
MOVL C01604 V=800.0 PL=0
MOVL C01605 V=800.0 PL=0
MOVL C01606 V=800.0 PL=0
MOVL C01607 V=800.0 PL=0
MOVL C01608 V=800.0 PL=0
MOVL C01609 V=800.0 PL=0
MOVL C01610 V=800.0 PL=0
MOVL C01611 V=800.0 PL=0
MOVL C01612 V=800.0 PL=0
MOVL C01613 V=800.0 PL=0
MOVL C01614 V=800.0 PL=0
MOVL C01615 V=800.0 PL=0
MOVL C01616 V=800.0 PL=0
MOVL C01617 V=800.0 PL=0
MOVL C01618 V=800.0 PL=0
MOVL C01619 V=800.0 PL=0
MOVL C01620 V=800.0 PL=0
MOVL C01621 V=800.0 PL=0
MOVL C01622 V=800.0 PL=0
MOVL C01623 V=800.0 PL=0
MOVL C01624 V=800.0 PL=0
MOVL C01625 V=800.0 PL=0
MOVL C01626 V=800.0 PL=0
MOVL C01627 V=800.0 PL=0
MOVL C01628 V=800.0 PL=0
MOVL C01629 V=800.0 PL=0
MOVL C01630 V=800.0 PL=0
MOVL C01631 V=800.0 PL=0
MOVL C01632 V=800.0 PL=0
MOVL C01633 V=800.0 PL=0
MOVL C01634 V=800.0 PL=0
MOVL C01635 V=800.0 PL=0
MOVL C01636 V=800.0 PL=0
MOVL C01637 V=800.0 PL=0
MOVL C01638 V=800.0 PL=0
MOVL C01639 V=800.0 PL=0
MOVL C01640 V=800.0 PL=0
MOVL C01641 V=800.0 PL=0
MOVL C01642 V=800.0 PL=0
MOVL C01643 V=800.0 PL=0
MOVL C01644 V=800.0 PL=0
MOVL C01645 V=800.0 PL=0
MOVL C01646 V=800.0 PL=0
MOVL C01647 V=800.0 PL=0
MOVL C01648 V=800.0 PL=0
MOVL C01649 V=800.0 PL=0
MOVL C01650 V=800.0 PL=0
MOVL C01651 V=800.0 PL=0
MOVL C01652 V=800.0 PL=0
MOVL C01653 V=800.0 PL=0
MOVL C01654 V=800.0 PL=0
MOVL C01655 V=800.0 PL=0
MOVL C01656 V=800.0 PL=0
MOVL C01657 V=800.0 PL=0
MOVL C01658 V=800.0 PL=0
MOVL C01659 V=800.0 PL=0
MOVL C01660 V=800.0 PL=0
MOVL C01661 V=800.0 PL=0
MOVL C01662 V=800.0 PL=0
MOVL C01663 V=800.0 PL=0
MOVL C01664 V=800.0 PL=0
MOVL C01665 V=800.0 PL=0
MOVL C01666 V=800.0 PL=0
MOVL C01667 V=800.0 PL=0
MOVL C01668 V=800.0 PL=0
MOVL C01669 V=800.0 PL=0
MOVL C01670 V=800.0 PL=0
MOVL C01671 V=800.0 PL=0
MOVL C01672 V=800.0 PL=0
MOVL C01673 V=800.0 PL=0
MOVL C01674 V=800.0 PL=0
MOVL C01675 V=800.0 PL=0
MOVL C01676 V=800.0 PL=0
MOVL C01677 V=800.0 PL=0
MOVL C01678 V=800.0 PL=0
MOVL C01679 V=800.0 PL=0
MOVL C01680 V=800.0 PL=0
MOVL C01681 V=800.0 PL=0
MOVL C01682 V=800.0 PL=0
MOVL C01683 V=800.0 PL=0
MOVL C01684 V=800.0 PL=0
MOVL C01685 V=800.0 PL=0
MOVL C01686 V=800.0 PL=0
MOVL C01687 V=800.0 PL=0
MOVL C01688 V=800.0 PL=0
MOVL C01689 V=800.0 PL=0
MOVL C01690 V=800.0 PL=0
MOVL C01691 V=800.0 PL=0
MOVL C01692 V=800.0 PL=0
MOVL C01693 V=800.0 PL=0
MOVL C01694 V=800.0 PL=0
MOVL C01695 V=800.0 PL=0
MOVL C01696 V=800.0 PL=0
MOVL C01697 V=800.0 PL=0
MOVL C01698 V=800.0 PL=0
MOVL C01699 V=800.0 PL=0
MOVL C01700 V=800.0 PL=0
MOVL C01701 V=800.0 PL=0
MOVL C01702 V=800.0 PL=0
MOVL C01703 V=800.0 PL=0
MOVL C01704 V=800.0 PL=0
MOVL C01705 V=800.0 PL=0
MOVL C01706 V=800.0 PL=0
MOVL C01707 V=800.0 PL=0
MOVL C01708 V=800.0 PL=0
MOVL C01709 V=800.0 PL=0
MOVL C01710 V=800.0 PL=0
MOVL C01711 V=800.0 PL=0
MOVL C01712 V=800.0 PL=0
MOVL C01713 V=800.0 PL=0
MOVL C01714 V=800.0 PL=0
MOVL C01715 V=800.0 PL=0
MOVL C01716 V=800.0 PL=0
MOVL C01717 V=800.0 PL=0
MOVL C01718 V=800.0 PL=0
MOVL C01719 V=800.0 PL=0
MOVL C01720 V=800.0 PL=0
MOVL C01721 V=800.0 PL=0
MOVL C01722 V=800.0 PL=0
MOVL C01723 V=800.0 PL=0
MOVL C01724 V=800.0 PL=0
MOVL C01725 V=800.0 PL=0
MOVL C01726 V=800.0 PL=0
MOVL C01727 V=800.0 PL=0
MOVL C01728 V=800.0 PL=0
MOVL C01729 V=800.0 PL=0
MOVL C01730 V=800.0 PL=0
MOVL C01731 V=800.0 PL=0
MOVL C01732 V=800.0 PL=0
MOVL C01733 V=800.0 PL=0
MOVL C01734 V=800.0 PL=0
MOVL C01735 V=800.0 PL=0
MOVL C01736 V=800.0 PL=0
MOVL C01737 V=800.0 PL=0
MOVL C01738 V=800.0 PL=0
MOVL C01739 V=800.0 PL=0
MOVL C01740 V=800.0 PL=0
MOVL C01741 V=800.0 PL=0
MOVL C01742 V=800.0 PL=0
MOVL C01743 V=800.0 PL=0
MOVL C01744 V=800.0 PL=0
MOVL C01745 V=800.0 PL=0
MOVL C01746 V=800.0 PL=0
MOVL C01747 V=800.0 PL=0
MOVL C01748 V=800.0 PL=0
MOVL C01749 V=800.0 PL=0
MOVL C01750 V=800.0 PL=0
MOVL C01751 V=800.0 PL=0
MOVL C01752 V=800.0 PL=0
MOVL C01753 V=800.0 PL=0
MOVL C01754 V=800.0 PL=0
MOVL C01755 V=800.0 PL=0
MOVL C01756 V=800.0 PL=0
MOVL C01757 V=800.0 PL=0
MOVL C01758 V=800.0 PL=0
MOVL C01759 V=800.0 PL=0
MOVL C01760 V=800.0 PL=0
MOVL C01761 V=800.0 PL=0
MOVL C01762 V=800.0 PL=0
MOVL C01763 V=800.0 PL=0
MOVL C01764 V=800.0 PL=0
MOVL C01765 V=800.0 PL=0
MOVL C01766 V=800.0 PL=0
MOVL C01767 V=800.0 PL=0
MOVL C01768 V=800.0 PL=0
MOVL C01769 V=800.0 PL=0
MOVL C01770 V=800.0 PL=0
MOVL C01771 V=800.0 PL=0
MOVL C01772 V=800.0 PL=0
MOVL C01773 V=800.0 PL=0
MOVL C01774 V=800.0 PL=0
MOVL C01775 V=800.0 PL=0
MOVL C01776 V=800.0 PL=0
MOVL C01777 V=800.0 PL=0
MOVL C01778 V=800.0 PL=0
MOVL C01779 V=800.0 PL=0
MOVL C01780 V=800.0 PL=0
MOVL C01781 V=800.0 PL=0
MOVL C01782 V=800.0 PL=0
MOVL C01783 V=800.0 PL=0
MOVL C01784 V=800.0 PL=0
MOVL C01785 V=800.0 PL=0
MOVL C01786 V=800.0 PL=0
MOVL C01787 V=800.0 PL=0
MOVL C01788 V=800.0 PL=0
MOVL C01789 V=800.0 PL=0
MOVL C01790 V=800.0 PL=0
MOVL C01791 V=800.0 PL=0
MOVL C01792 V=800.0 PL=0
MOVL C01793 V=800.0 PL=0
MOVL C01794 V=800.0 PL=0
MOVL C01795 V=800.0 PL=0
MOVL C01796 V=800.0 PL=0
MOVL C01797 V=800.0 PL=0
MOVL C01798 V=800.0 PL=0
MOVL C01799 V=800.0 PL=0
MOVL C01800 V=800.0 PL=0
MOVL C01801 V=800.0 PL=0
MOVL C01802 V=800.0 PL=0
MOVL C01803 V=800.0 PL=0
MOVL C01804 V=800.0 PL=0
MOVL C01805 V=800.0 PL=0
MOVL C01806 V=800.0 PL=0
MOVL C01807 V=800.0 PL=0
MOVL C01808 V=800.0 PL=0
MOVL C01809 V=800.0 PL=0
MOVL C01810 V=800.0 PL=0
MOVL C01811 V=800.0 PL=0
MOVL C01812 V=800.0 PL=0
MOVL C01813 V=800.0 PL=0
MOVL C01814 V=800.0 PL=0
MOVL C01815 V=800.0 PL=0
MOVL C01816 V=800.0 PL=0
MOVL C01817 V=800.0 PL=0
MOVL C01818 V=800.0 PL=0
MOVL C01819 V=800.0 PL=0
MOVL C01820 V=800.0 PL=0
MOVL C01821 V=800.0 PL=0
MOVL C01822 V=800.0 PL=0
MOVL C01823 V=800.0 PL=0
MOVL C01824 V=800.0 PL=0
MOVL C01825 V=800.0 PL=0
MOVL C01826 V=800.0 PL=0
MOVL C01827 V=800.0 PL=0
MOVL C01828 V=800.0 PL=0
MOVL C01829 V=800.0 PL=0
MOVL C01830 V=800.0 PL=0
MOVL C01831 V=800.0 PL=0
MOVL C01832 V=800.0 PL=0
MOVL C01833 V=800.0 PL=0
MOVL C01834 V=800.0 PL=0
MOVL C01835 V=800.0 PL=0
MOVL C01836 V=800.0 PL=0
MOVL C01837 V=800.0 PL=0
MOVL C01838 V=800.0 PL=0
MOVL C01839 V=800.0 PL=0
MOVL C01840 V=800.0 PL=0
MOVL C01841 V=800.0 PL=0
MOVL C01842 V=800.0 PL=0
MOVL C01843 V=800.0 PL=0
MOVL C01844 V=800.0 PL=0
MOVL C01845 V=800.0 PL=0
MOVL C01846 V=800.0 PL=0
MOVL C01847 V=800.0 PL=0
MOVL C01848 V=800.0 PL=0
MOVL C01849 V=800.0 PL=0
MOVL C01850 V=800.0 PL=0
MOVL C01851 V=800.0 PL=0
MOVL C01852 V=800.0 PL=0
MOVL C01853 V=800.0 PL=0
MOVL C01854 V=800.0 PL=0
MOVL C01855 V=800.0 PL=0
